   // UNICODE_TO_GBK[14826] := 16#6828;
   // UNICODE_TO_GBK[14827] := 16#96E6;
   // UNICODE_TO_GBK[14828] := 16#6829;
   // UNICODE_TO_GBK[14829] := 16#E8F2;
   // UNICODE_TO_GBK[14830] := 16#682A;
   // UNICODE_TO_GBK[14831] := 16#D6EA;
   // UNICODE_TO_GBK[14832] := 16#682B;
   // UNICODE_TO_GBK[14833] := 16#96E7;
   // UNICODE_TO_GBK[14834] := 16#682C;
   // UNICODE_TO_GBK[14835] := 16#96E8;
   // UNICODE_TO_GBK[14836] := 16#682D;
   // UNICODE_TO_GBK[14837] := 16#96E9;
   // UNICODE_TO_GBK[14838] := 16#682E;
   // UNICODE_TO_GBK[14839] := 16#96EA;
   // UNICODE_TO_GBK[14840] := 16#682F;
   // UNICODE_TO_GBK[14841] := 16#96EB;
   // UNICODE_TO_GBK[14842] := 16#6830;
   // UNICODE_TO_GBK[14843] := 16#96EC;
   // UNICODE_TO_GBK[14844] := 16#6831;
   // UNICODE_TO_GBK[14845] := 16#96ED;
   // UNICODE_TO_GBK[14846] := 16#6832;
   // UNICODE_TO_GBK[14847] := 16#E8E0;
   // UNICODE_TO_GBK[14848] := 16#6833;
   // UNICODE_TO_GBK[14849] := 16#E8E1;
   // UNICODE_TO_GBK[14850] := 16#6834;
   // UNICODE_TO_GBK[14851] := 16#96EE;
   // UNICODE_TO_GBK[14852] := 16#6835;
   // UNICODE_TO_GBK[14853] := 16#96EF;
   // UNICODE_TO_GBK[14854] := 16#6836;
   // UNICODE_TO_GBK[14855] := 16#96F0;
   // UNICODE_TO_GBK[14856] := 16#6837;
   // UNICODE_TO_GBK[14857] := 16#D1F9;
   // UNICODE_TO_GBK[14858] := 16#6838;
   // UNICODE_TO_GBK[14859] := 16#BACB;
   // UNICODE_TO_GBK[14860] := 16#6839;
   // UNICODE_TO_GBK[14861] := 16#B8F9;
   // UNICODE_TO_GBK[14862] := 16#683A;
   // UNICODE_TO_GBK[14863] := 16#96F1;
   // UNICODE_TO_GBK[14864] := 16#683B;
   // UNICODE_TO_GBK[14865] := 16#96F2;
   // UNICODE_TO_GBK[14866] := 16#683C;
   // UNICODE_TO_GBK[14867] := 16#B8F1;
   // UNICODE_TO_GBK[14868] := 16#683D;
   // UNICODE_TO_GBK[14869] := 16#D4D4;
   // UNICODE_TO_GBK[14870] := 16#683E;
   // UNICODE_TO_GBK[14871] := 16#E8EF;
   // UNICODE_TO_GBK[14872] := 16#683F;
   // UNICODE_TO_GBK[14873] := 16#96F3;
   // UNICODE_TO_GBK[14874] := 16#6840;
   // UNICODE_TO_GBK[14875] := 16#E8EE;
   // UNICODE_TO_GBK[14876] := 16#6841;
   // UNICODE_TO_GBK[14877] := 16#E8EC;
   // UNICODE_TO_GBK[14878] := 16#6842;
   // UNICODE_TO_GBK[14879] := 16#B9F0;
   // UNICODE_TO_GBK[14880] := 16#6843;
   // UNICODE_TO_GBK[14881] := 16#CCD2;
   // UNICODE_TO_GBK[14882] := 16#6844;
   // UNICODE_TO_GBK[14883] := 16#E8E6;
   // UNICODE_TO_GBK[14884] := 16#6845;
   // UNICODE_TO_GBK[14885] := 16#CEA6;
   // UNICODE_TO_GBK[14886] := 16#6846;
   // UNICODE_TO_GBK[14887] := 16#BFF2;
   // UNICODE_TO_GBK[14888] := 16#6847;
   // UNICODE_TO_GBK[14889] := 16#96F4;
   // UNICODE_TO_GBK[14890] := 16#6848;
   // UNICODE_TO_GBK[14891] := 16#B0B8;
   // UNICODE_TO_GBK[14892] := 16#6849;
   // UNICODE_TO_GBK[14893] := 16#E8F1;
   // UNICODE_TO_GBK[14894] := 16#684A;
   // UNICODE_TO_GBK[14895] := 16#E8F0;
   // UNICODE_TO_GBK[14896] := 16#684B;
   // UNICODE_TO_GBK[14897] := 16#96F5;
   // UNICODE_TO_GBK[14898] := 16#684C;
   // UNICODE_TO_GBK[14899] := 16#D7C0;
   // UNICODE_TO_GBK[14900] := 16#684D;
   // UNICODE_TO_GBK[14901] := 16#96F6;
   // UNICODE_TO_GBK[14902] := 16#684E;
   // UNICODE_TO_GBK[14903] := 16#E8E4;
   // UNICODE_TO_GBK[14904] := 16#684F;
   // UNICODE_TO_GBK[14905] := 16#96F7;
   // UNICODE_TO_GBK[14906] := 16#6850;
   // UNICODE_TO_GBK[14907] := 16#CDA9;
   // UNICODE_TO_GBK[14908] := 16#6851;
   // UNICODE_TO_GBK[14909] := 16#C9A3;
   // UNICODE_TO_GBK[14910] := 16#6852;
   // UNICODE_TO_GBK[14911] := 16#96F8;
   // UNICODE_TO_GBK[14912] := 16#6853;
   // UNICODE_TO_GBK[14913] := 16#BBB8;
   // UNICODE_TO_GBK[14914] := 16#6854;
   // UNICODE_TO_GBK[14915] := 16#BDDB;
   // UNICODE_TO_GBK[14916] := 16#6855;
   // UNICODE_TO_GBK[14917] := 16#E8EA;
   // UNICODE_TO_GBK[14918] := 16#6856;
   // UNICODE_TO_GBK[14919] := 16#96F9;
   // UNICODE_TO_GBK[14920] := 16#6857;
   // UNICODE_TO_GBK[14921] := 16#96FA;
   // UNICODE_TO_GBK[14922] := 16#6858;
   // UNICODE_TO_GBK[14923] := 16#96FB;
   // UNICODE_TO_GBK[14924] := 16#6859;
   // UNICODE_TO_GBK[14925] := 16#96FC;
   // UNICODE_TO_GBK[14926] := 16#685A;
   // UNICODE_TO_GBK[14927] := 16#96FD;
   // UNICODE_TO_GBK[14928] := 16#685B;
   // UNICODE_TO_GBK[14929] := 16#96FE;
   // UNICODE_TO_GBK[14930] := 16#685C;
   // UNICODE_TO_GBK[14931] := 16#9740;
   // UNICODE_TO_GBK[14932] := 16#685D;
   // UNICODE_TO_GBK[14933] := 16#9741;
   // UNICODE_TO_GBK[14934] := 16#685E;
   // UNICODE_TO_GBK[14935] := 16#9742;
   // UNICODE_TO_GBK[14936] := 16#685F;
   // UNICODE_TO_GBK[14937] := 16#9743;
   // UNICODE_TO_GBK[14938] := 16#6860;
   // UNICODE_TO_GBK[14939] := 16#E8E2;
   // UNICODE_TO_GBK[14940] := 16#6861;
   // UNICODE_TO_GBK[14941] := 16#E8E3;
   // UNICODE_TO_GBK[14942] := 16#6862;
   // UNICODE_TO_GBK[14943] := 16#E8E5;
   // UNICODE_TO_GBK[14944] := 16#6863;
   // UNICODE_TO_GBK[14945] := 16#B5B5;
   // UNICODE_TO_GBK[14946] := 16#6864;
   // UNICODE_TO_GBK[14947] := 16#E8E7;
   // UNICODE_TO_GBK[14948] := 16#6865;
   // UNICODE_TO_GBK[14949] := 16#C7C5;
   // UNICODE_TO_GBK[14950] := 16#6866;
   // UNICODE_TO_GBK[14951] := 16#E8EB;
   // UNICODE_TO_GBK[14952] := 16#6867;
   // UNICODE_TO_GBK[14953] := 16#E8ED;
   // UNICODE_TO_GBK[14954] := 16#6868;
   // UNICODE_TO_GBK[14955] := 16#BDB0;
   // UNICODE_TO_GBK[14956] := 16#6869;
   // UNICODE_TO_GBK[14957] := 16#D7AE;
   // UNICODE_TO_GBK[14958] := 16#686A;
   // UNICODE_TO_GBK[14959] := 16#9744;
   // UNICODE_TO_GBK[14960] := 16#686B;
   // UNICODE_TO_GBK[14961] := 16#E8F8;
   // UNICODE_TO_GBK[14962] := 16#686C;
   // UNICODE_TO_GBK[14963] := 16#9745;
   // UNICODE_TO_GBK[14964] := 16#686D;
   // UNICODE_TO_GBK[14965] := 16#9746;
   // UNICODE_TO_GBK[14966] := 16#686E;
   // UNICODE_TO_GBK[14967] := 16#9747;
   // UNICODE_TO_GBK[14968] := 16#686F;
   // UNICODE_TO_GBK[14969] := 16#9748;
   // UNICODE_TO_GBK[14970] := 16#6870;
   // UNICODE_TO_GBK[14971] := 16#9749;
   // UNICODE_TO_GBK[14972] := 16#6871;
   // UNICODE_TO_GBK[14973] := 16#974A;
   // UNICODE_TO_GBK[14974] := 16#6872;
   // UNICODE_TO_GBK[14975] := 16#974B;
   // UNICODE_TO_GBK[14976] := 16#6873;
   // UNICODE_TO_GBK[14977] := 16#974C;
   // UNICODE_TO_GBK[14978] := 16#6874;
   // UNICODE_TO_GBK[14979] := 16#E8F5;
   // UNICODE_TO_GBK[14980] := 16#6875;
   // UNICODE_TO_GBK[14981] := 16#974D;
   // UNICODE_TO_GBK[14982] := 16#6876;
   // UNICODE_TO_GBK[14983] := 16#CDB0;
   // UNICODE_TO_GBK[14984] := 16#6877;
   // UNICODE_TO_GBK[14985] := 16#E8F6;
   // UNICODE_TO_GBK[14986] := 16#6878;
   // UNICODE_TO_GBK[14987] := 16#974E;
   // UNICODE_TO_GBK[14988] := 16#6879;
   // UNICODE_TO_GBK[14989] := 16#974F;
   // UNICODE_TO_GBK[14990] := 16#687A;
   // UNICODE_TO_GBK[14991] := 16#9750;
   // UNICODE_TO_GBK[14992] := 16#687B;
   // UNICODE_TO_GBK[14993] := 16#9751;
   // UNICODE_TO_GBK[14994] := 16#687C;
   // UNICODE_TO_GBK[14995] := 16#9752;
   // UNICODE_TO_GBK[14996] := 16#687D;
   // UNICODE_TO_GBK[14997] := 16#9753;
   // UNICODE_TO_GBK[14998] := 16#687E;
   // UNICODE_TO_GBK[14999] := 16#9754;
   // UNICODE_TO_GBK[15000] := 16#687F;
   // UNICODE_TO_GBK[15001] := 16#9755;
   // UNICODE_TO_GBK[15002] := 16#6880;
   // UNICODE_TO_GBK[15003] := 16#9756;
   // UNICODE_TO_GBK[15004] := 16#6881;
   // UNICODE_TO_GBK[15005] := 16#C1BA;
   // UNICODE_TO_GBK[15006] := 16#6882;
   // UNICODE_TO_GBK[15007] := 16#9757;
   // UNICODE_TO_GBK[15008] := 16#6883;
   // UNICODE_TO_GBK[15009] := 16#E8E8;
   // UNICODE_TO_GBK[15010] := 16#6884;
   // UNICODE_TO_GBK[15011] := 16#9758;
   // UNICODE_TO_GBK[15012] := 16#6885;
   // UNICODE_TO_GBK[15013] := 16#C3B7;
   // UNICODE_TO_GBK[15014] := 16#6886;
   // UNICODE_TO_GBK[15015] := 16#B0F0;
   // UNICODE_TO_GBK[15016] := 16#6887;
   // UNICODE_TO_GBK[15017] := 16#9759;
   // UNICODE_TO_GBK[15018] := 16#6888;
   // UNICODE_TO_GBK[15019] := 16#975A;
   // UNICODE_TO_GBK[15020] := 16#6889;
   // UNICODE_TO_GBK[15021] := 16#975B;
   // UNICODE_TO_GBK[15022] := 16#688A;
   // UNICODE_TO_GBK[15023] := 16#975C;
   // UNICODE_TO_GBK[15024] := 16#688B;
   // UNICODE_TO_GBK[15025] := 16#975D;
   // UNICODE_TO_GBK[15026] := 16#688C;
   // UNICODE_TO_GBK[15027] := 16#975E;
   // UNICODE_TO_GBK[15028] := 16#688D;
   // UNICODE_TO_GBK[15029] := 16#975F;
   // UNICODE_TO_GBK[15030] := 16#688E;
   // UNICODE_TO_GBK[15031] := 16#9760;
   // UNICODE_TO_GBK[15032] := 16#688F;
   // UNICODE_TO_GBK[15033] := 16#E8F4;
   // UNICODE_TO_GBK[15034] := 16#6890;
   // UNICODE_TO_GBK[15035] := 16#9761;
   // UNICODE_TO_GBK[15036] := 16#6891;
   // UNICODE_TO_GBK[15037] := 16#9762;
   // UNICODE_TO_GBK[15038] := 16#6892;
   // UNICODE_TO_GBK[15039] := 16#9763;
   // UNICODE_TO_GBK[15040] := 16#6893;
   // UNICODE_TO_GBK[15041] := 16#E8F7;
   // UNICODE_TO_GBK[15042] := 16#6894;
   // UNICODE_TO_GBK[15043] := 16#9764;
   // UNICODE_TO_GBK[15044] := 16#6895;
   // UNICODE_TO_GBK[15045] := 16#9765;
   // UNICODE_TO_GBK[15046] := 16#6896;
   // UNICODE_TO_GBK[15047] := 16#9766;
   // UNICODE_TO_GBK[15048] := 16#6897;
   // UNICODE_TO_GBK[15049] := 16#B9A3;
   // UNICODE_TO_GBK[15050] := 16#6898;
   // UNICODE_TO_GBK[15051] := 16#9767;
   // UNICODE_TO_GBK[15052] := 16#6899;
   // UNICODE_TO_GBK[15053] := 16#9768;
   // UNICODE_TO_GBK[15054] := 16#689A;
   // UNICODE_TO_GBK[15055] := 16#9769;
   // UNICODE_TO_GBK[15056] := 16#689B;
   // UNICODE_TO_GBK[15057] := 16#976A;
   // UNICODE_TO_GBK[15058] := 16#689C;
   // UNICODE_TO_GBK[15059] := 16#976B;
   // UNICODE_TO_GBK[15060] := 16#689D;
   // UNICODE_TO_GBK[15061] := 16#976C;
   // UNICODE_TO_GBK[15062] := 16#689E;
   // UNICODE_TO_GBK[15063] := 16#976D;
   // UNICODE_TO_GBK[15064] := 16#689F;
   // UNICODE_TO_GBK[15065] := 16#976E;
   // UNICODE_TO_GBK[15066] := 16#68A0;
   // UNICODE_TO_GBK[15067] := 16#976F;
   // UNICODE_TO_GBK[15068] := 16#68A1;
   // UNICODE_TO_GBK[15069] := 16#9770;
   // UNICODE_TO_GBK[15070] := 16#68A2;
   // UNICODE_TO_GBK[15071] := 16#C9D2;
   // UNICODE_TO_GBK[15072] := 16#68A3;
   // UNICODE_TO_GBK[15073] := 16#9771;
   // UNICODE_TO_GBK[15074] := 16#68A4;
   // UNICODE_TO_GBK[15075] := 16#9772;
   // UNICODE_TO_GBK[15076] := 16#68A5;
   // UNICODE_TO_GBK[15077] := 16#9773;
   // UNICODE_TO_GBK[15078] := 16#68A6;
   // UNICODE_TO_GBK[15079] := 16#C3CE;
   // UNICODE_TO_GBK[15080] := 16#68A7;
   // UNICODE_TO_GBK[15081] := 16#CEE0;
   // UNICODE_TO_GBK[15082] := 16#68A8;
   // UNICODE_TO_GBK[15083] := 16#C0E6;
   // UNICODE_TO_GBK[15084] := 16#68A9;
   // UNICODE_TO_GBK[15085] := 16#9774;
   // UNICODE_TO_GBK[15086] := 16#68AA;
   // UNICODE_TO_GBK[15087] := 16#9775;
   // UNICODE_TO_GBK[15088] := 16#68AB;
   // UNICODE_TO_GBK[15089] := 16#9776;
   // UNICODE_TO_GBK[15090] := 16#68AC;
   // UNICODE_TO_GBK[15091] := 16#9777;
   // UNICODE_TO_GBK[15092] := 16#68AD;
   // UNICODE_TO_GBK[15093] := 16#CBF3;
   // UNICODE_TO_GBK[15094] := 16#68AE;
   // UNICODE_TO_GBK[15095] := 16#9778;
   // UNICODE_TO_GBK[15096] := 16#68AF;
   // UNICODE_TO_GBK[15097] := 16#CCDD;
   // UNICODE_TO_GBK[15098] := 16#68B0;
   // UNICODE_TO_GBK[15099] := 16#D0B5;
   // UNICODE_TO_GBK[15100] := 16#68B1;
   // UNICODE_TO_GBK[15101] := 16#9779;
   // UNICODE_TO_GBK[15102] := 16#68B2;
   // UNICODE_TO_GBK[15103] := 16#977A;
   // UNICODE_TO_GBK[15104] := 16#68B3;
   // UNICODE_TO_GBK[15105] := 16#CAE1;
   // UNICODE_TO_GBK[15106] := 16#68B4;
   // UNICODE_TO_GBK[15107] := 16#977B;
   // UNICODE_TO_GBK[15108] := 16#68B5;
   // UNICODE_TO_GBK[15109] := 16#E8F3;
   // UNICODE_TO_GBK[15110] := 16#68B6;
   // UNICODE_TO_GBK[15111] := 16#977C;
   // UNICODE_TO_GBK[15112] := 16#68B7;
   // UNICODE_TO_GBK[15113] := 16#977D;
   // UNICODE_TO_GBK[15114] := 16#68B8;
   // UNICODE_TO_GBK[15115] := 16#977E;
   // UNICODE_TO_GBK[15116] := 16#68B9;
   // UNICODE_TO_GBK[15117] := 16#9780;
   // UNICODE_TO_GBK[15118] := 16#68BA;
   // UNICODE_TO_GBK[15119] := 16#9781;
   // UNICODE_TO_GBK[15120] := 16#68BB;
   // UNICODE_TO_GBK[15121] := 16#9782;
   // UNICODE_TO_GBK[15122] := 16#68BC;
   // UNICODE_TO_GBK[15123] := 16#9783;
   // UNICODE_TO_GBK[15124] := 16#68BD;
   // UNICODE_TO_GBK[15125] := 16#9784;
   // UNICODE_TO_GBK[15126] := 16#68BE;
   // UNICODE_TO_GBK[15127] := 16#9785;
   // UNICODE_TO_GBK[15128] := 16#68BF;
   // UNICODE_TO_GBK[15129] := 16#9786;
   // UNICODE_TO_GBK[15130] := 16#68C0;
   // UNICODE_TO_GBK[15131] := 16#BCEC;
   // UNICODE_TO_GBK[15132] := 16#68C1;
   // UNICODE_TO_GBK[15133] := 16#9787;
   // UNICODE_TO_GBK[15134] := 16#68C2;
   // UNICODE_TO_GBK[15135] := 16#E8F9;
   // UNICODE_TO_GBK[15136] := 16#68C3;
   // UNICODE_TO_GBK[15137] := 16#9788;
   // UNICODE_TO_GBK[15138] := 16#68C4;
   // UNICODE_TO_GBK[15139] := 16#9789;
   // UNICODE_TO_GBK[15140] := 16#68C5;
   // UNICODE_TO_GBK[15141] := 16#978A;
   // UNICODE_TO_GBK[15142] := 16#68C6;
   // UNICODE_TO_GBK[15143] := 16#978B;
   // UNICODE_TO_GBK[15144] := 16#68C7;
   // UNICODE_TO_GBK[15145] := 16#978C;
   // UNICODE_TO_GBK[15146] := 16#68C8;
   // UNICODE_TO_GBK[15147] := 16#978D;
   // UNICODE_TO_GBK[15148] := 16#68C9;
   // UNICODE_TO_GBK[15149] := 16#C3DE;
   // UNICODE_TO_GBK[15150] := 16#68CA;
   // UNICODE_TO_GBK[15151] := 16#978E;
   // UNICODE_TO_GBK[15152] := 16#68CB;
   // UNICODE_TO_GBK[15153] := 16#C6E5;
   // UNICODE_TO_GBK[15154] := 16#68CC;
   // UNICODE_TO_GBK[15155] := 16#978F;
   // UNICODE_TO_GBK[15156] := 16#68CD;
   // UNICODE_TO_GBK[15157] := 16#B9F7;
   // UNICODE_TO_GBK[15158] := 16#68CE;
   // UNICODE_TO_GBK[15159] := 16#9790;
   // UNICODE_TO_GBK[15160] := 16#68CF;
   // UNICODE_TO_GBK[15161] := 16#9791;
   // UNICODE_TO_GBK[15162] := 16#68D0;
   // UNICODE_TO_GBK[15163] := 16#9792;
   // UNICODE_TO_GBK[15164] := 16#68D1;
   // UNICODE_TO_GBK[15165] := 16#9793;
   // UNICODE_TO_GBK[15166] := 16#68D2;
   // UNICODE_TO_GBK[15167] := 16#B0F4;
   // UNICODE_TO_GBK[15168] := 16#68D3;
   // UNICODE_TO_GBK[15169] := 16#9794;
   // UNICODE_TO_GBK[15170] := 16#68D4;
   // UNICODE_TO_GBK[15171] := 16#9795;
   // UNICODE_TO_GBK[15172] := 16#68D5;
   // UNICODE_TO_GBK[15173] := 16#D7D8;
   // UNICODE_TO_GBK[15174] := 16#68D6;
   // UNICODE_TO_GBK[15175] := 16#9796;
   // UNICODE_TO_GBK[15176] := 16#68D7;
   // UNICODE_TO_GBK[15177] := 16#9797;
   // UNICODE_TO_GBK[15178] := 16#68D8;
   // UNICODE_TO_GBK[15179] := 16#BCAC;
   // UNICODE_TO_GBK[15180] := 16#68D9;
   // UNICODE_TO_GBK[15181] := 16#9798;
   // UNICODE_TO_GBK[15182] := 16#68DA;
   // UNICODE_TO_GBK[15183] := 16#C5EF;
   // UNICODE_TO_GBK[15184] := 16#68DB;
   // UNICODE_TO_GBK[15185] := 16#9799;
   // UNICODE_TO_GBK[15186] := 16#68DC;
   // UNICODE_TO_GBK[15187] := 16#979A;
   // UNICODE_TO_GBK[15188] := 16#68DD;
   // UNICODE_TO_GBK[15189] := 16#979B;
   // UNICODE_TO_GBK[15190] := 16#68DE;
   // UNICODE_TO_GBK[15191] := 16#979C;
   // UNICODE_TO_GBK[15192] := 16#68DF;
   // UNICODE_TO_GBK[15193] := 16#979D;
   // UNICODE_TO_GBK[15194] := 16#68E0;
   // UNICODE_TO_GBK[15195] := 16#CCC4;
   // UNICODE_TO_GBK[15196] := 16#68E1;
   // UNICODE_TO_GBK[15197] := 16#979E;
   // UNICODE_TO_GBK[15198] := 16#68E2;
   // UNICODE_TO_GBK[15199] := 16#979F;
   // UNICODE_TO_GBK[15200] := 16#68E3;
   // UNICODE_TO_GBK[15201] := 16#E9A6;
   // UNICODE_TO_GBK[15202] := 16#68E4;
   // UNICODE_TO_GBK[15203] := 16#97A0;
   // UNICODE_TO_GBK[15204] := 16#68E5;
   // UNICODE_TO_GBK[15205] := 16#97A1;
   // UNICODE_TO_GBK[15206] := 16#68E6;
   // UNICODE_TO_GBK[15207] := 16#97A2;
   // UNICODE_TO_GBK[15208] := 16#68E7;
   // UNICODE_TO_GBK[15209] := 16#97A3;
   // UNICODE_TO_GBK[15210] := 16#68E8;
   // UNICODE_TO_GBK[15211] := 16#97A4;
   // UNICODE_TO_GBK[15212] := 16#68E9;
   // UNICODE_TO_GBK[15213] := 16#97A5;
   // UNICODE_TO_GBK[15214] := 16#68EA;
   // UNICODE_TO_GBK[15215] := 16#97A6;
   // UNICODE_TO_GBK[15216] := 16#68EB;
   // UNICODE_TO_GBK[15217] := 16#97A7;
   // UNICODE_TO_GBK[15218] := 16#68EC;
   // UNICODE_TO_GBK[15219] := 16#97A8;
   // UNICODE_TO_GBK[15220] := 16#68ED;
   // UNICODE_TO_GBK[15221] := 16#97A9;
   // UNICODE_TO_GBK[15222] := 16#68EE;
   // UNICODE_TO_GBK[15223] := 16#C9AD;
   // UNICODE_TO_GBK[15224] := 16#68EF;
   // UNICODE_TO_GBK[15225] := 16#97AA;
   // UNICODE_TO_GBK[15226] := 16#68F0;
   // UNICODE_TO_GBK[15227] := 16#E9A2;
   // UNICODE_TO_GBK[15228] := 16#68F1;
   // UNICODE_TO_GBK[15229] := 16#C0E2;
   // UNICODE_TO_GBK[15230] := 16#68F2;
   // UNICODE_TO_GBK[15231] := 16#97AB;
   // UNICODE_TO_GBK[15232] := 16#68F3;
   // UNICODE_TO_GBK[15233] := 16#97AC;
   // UNICODE_TO_GBK[15234] := 16#68F4;
   // UNICODE_TO_GBK[15235] := 16#97AD;
   // UNICODE_TO_GBK[15236] := 16#68F5;
   // UNICODE_TO_GBK[15237] := 16#BFC3;
   // UNICODE_TO_GBK[15238] := 16#68F6;
   // UNICODE_TO_GBK[15239] := 16#97AE;
   // UNICODE_TO_GBK[15240] := 16#68F7;
   // UNICODE_TO_GBK[15241] := 16#97AF;
   // UNICODE_TO_GBK[15242] := 16#68F8;
   // UNICODE_TO_GBK[15243] := 16#97B0;
   // UNICODE_TO_GBK[15244] := 16#68F9;
   // UNICODE_TO_GBK[15245] := 16#E8FE;
   // UNICODE_TO_GBK[15246] := 16#68FA;
   // UNICODE_TO_GBK[15247] := 16#B9D7;
   // UNICODE_TO_GBK[15248] := 16#68FB;
   // UNICODE_TO_GBK[15249] := 16#97B1;
   // UNICODE_TO_GBK[15250] := 16#68FC;
   // UNICODE_TO_GBK[15251] := 16#E8FB;
   // UNICODE_TO_GBK[15252] := 16#68FD;
   // UNICODE_TO_GBK[15253] := 16#97B2;
   // UNICODE_TO_GBK[15254] := 16#68FE;
   // UNICODE_TO_GBK[15255] := 16#97B3;
   // UNICODE_TO_GBK[15256] := 16#68FF;
   // UNICODE_TO_GBK[15257] := 16#97B4;
   // UNICODE_TO_GBK[15258] := 16#6900;
   // UNICODE_TO_GBK[15259] := 16#97B5;
   // UNICODE_TO_GBK[15260] := 16#6901;
   // UNICODE_TO_GBK[15261] := 16#E9A4;
   // UNICODE_TO_GBK[15262] := 16#6902;
   // UNICODE_TO_GBK[15263] := 16#97B6;
   // UNICODE_TO_GBK[15264] := 16#6903;
   // UNICODE_TO_GBK[15265] := 16#97B7;
   // UNICODE_TO_GBK[15266] := 16#6904;
   // UNICODE_TO_GBK[15267] := 16#97B8;
   // UNICODE_TO_GBK[15268] := 16#6905;
   // UNICODE_TO_GBK[15269] := 16#D2CE;
   // UNICODE_TO_GBK[15270] := 16#6906;
   // UNICODE_TO_GBK[15271] := 16#97B9;
   // UNICODE_TO_GBK[15272] := 16#6907;
   // UNICODE_TO_GBK[15273] := 16#97BA;
   // UNICODE_TO_GBK[15274] := 16#6908;
   // UNICODE_TO_GBK[15275] := 16#97BB;
   // UNICODE_TO_GBK[15276] := 16#6909;
   // UNICODE_TO_GBK[15277] := 16#97BC;
   // UNICODE_TO_GBK[15278] := 16#690A;
   // UNICODE_TO_GBK[15279] := 16#97BD;
   // UNICODE_TO_GBK[15280] := 16#690B;
   // UNICODE_TO_GBK[15281] := 16#E9A3;
   // UNICODE_TO_GBK[15282] := 16#690C;
   // UNICODE_TO_GBK[15283] := 16#97BE;
   // UNICODE_TO_GBK[15284] := 16#690D;
   // UNICODE_TO_GBK[15285] := 16#D6B2;
   // UNICODE_TO_GBK[15286] := 16#690E;
   // UNICODE_TO_GBK[15287] := 16#D7B5;
   // UNICODE_TO_GBK[15288] := 16#690F;
   // UNICODE_TO_GBK[15289] := 16#97BF;
   // UNICODE_TO_GBK[15290] := 16#6910;
   // UNICODE_TO_GBK[15291] := 16#E9A7;
   // UNICODE_TO_GBK[15292] := 16#6911;
   // UNICODE_TO_GBK[15293] := 16#97C0;
   // UNICODE_TO_GBK[15294] := 16#6912;
   // UNICODE_TO_GBK[15295] := 16#BDB7;
   // UNICODE_TO_GBK[15296] := 16#6913;
   // UNICODE_TO_GBK[15297] := 16#97C1;
   // UNICODE_TO_GBK[15298] := 16#6914;
   // UNICODE_TO_GBK[15299] := 16#97C2;
   // UNICODE_TO_GBK[15300] := 16#6915;
   // UNICODE_TO_GBK[15301] := 16#97C3;
   // UNICODE_TO_GBK[15302] := 16#6916;
   // UNICODE_TO_GBK[15303] := 16#97C4;
   // UNICODE_TO_GBK[15304] := 16#6917;
   // UNICODE_TO_GBK[15305] := 16#97C5;
   // UNICODE_TO_GBK[15306] := 16#6918;
   // UNICODE_TO_GBK[15307] := 16#97C6;
   // UNICODE_TO_GBK[15308] := 16#6919;
   // UNICODE_TO_GBK[15309] := 16#97C7;
   // UNICODE_TO_GBK[15310] := 16#691A;
   // UNICODE_TO_GBK[15311] := 16#97C8;
   // UNICODE_TO_GBK[15312] := 16#691B;
   // UNICODE_TO_GBK[15313] := 16#97C9;
   // UNICODE_TO_GBK[15314] := 16#691C;
   // UNICODE_TO_GBK[15315] := 16#97CA;
   // UNICODE_TO_GBK[15316] := 16#691D;
   // UNICODE_TO_GBK[15317] := 16#97CB;
   // UNICODE_TO_GBK[15318] := 16#691E;
   // UNICODE_TO_GBK[15319] := 16#97CC;
   // UNICODE_TO_GBK[15320] := 16#691F;
   // UNICODE_TO_GBK[15321] := 16#E8FC;
   // UNICODE_TO_GBK[15322] := 16#6920;
   // UNICODE_TO_GBK[15323] := 16#E8FD;
   // UNICODE_TO_GBK[15324] := 16#6921;
   // UNICODE_TO_GBK[15325] := 16#97CD;
   // UNICODE_TO_GBK[15326] := 16#6922;
   // UNICODE_TO_GBK[15327] := 16#97CE;
   // UNICODE_TO_GBK[15328] := 16#6923;
   // UNICODE_TO_GBK[15329] := 16#97CF;
   // UNICODE_TO_GBK[15330] := 16#6924;
   // UNICODE_TO_GBK[15331] := 16#E9A1;
   // UNICODE_TO_GBK[15332] := 16#6925;
   // UNICODE_TO_GBK[15333] := 16#97D0;
   // UNICODE_TO_GBK[15334] := 16#6926;
   // UNICODE_TO_GBK[15335] := 16#97D1;
   // UNICODE_TO_GBK[15336] := 16#6927;
   // UNICODE_TO_GBK[15337] := 16#97D2;
   // UNICODE_TO_GBK[15338] := 16#6928;
   // UNICODE_TO_GBK[15339] := 16#97D3;
   // UNICODE_TO_GBK[15340] := 16#6929;
   // UNICODE_TO_GBK[15341] := 16#97D4;
   // UNICODE_TO_GBK[15342] := 16#692A;
   // UNICODE_TO_GBK[15343] := 16#97D5;
   // UNICODE_TO_GBK[15344] := 16#692B;
   // UNICODE_TO_GBK[15345] := 16#97D6;
   // UNICODE_TO_GBK[15346] := 16#692C;
   // UNICODE_TO_GBK[15347] := 16#97D7;
   // UNICODE_TO_GBK[15348] := 16#692D;
   // UNICODE_TO_GBK[15349] := 16#CDD6;
   // UNICODE_TO_GBK[15350] := 16#692E;
   // UNICODE_TO_GBK[15351] := 16#97D8;
   // UNICODE_TO_GBK[15352] := 16#692F;
   // UNICODE_TO_GBK[15353] := 16#97D9;
   // UNICODE_TO_GBK[15354] := 16#6930;
   // UNICODE_TO_GBK[15355] := 16#D2AC;
   // UNICODE_TO_GBK[15356] := 16#6931;
   // UNICODE_TO_GBK[15357] := 16#97DA;
   // UNICODE_TO_GBK[15358] := 16#6932;
   // UNICODE_TO_GBK[15359] := 16#97DB;
   // UNICODE_TO_GBK[15360] := 16#6933;
   // UNICODE_TO_GBK[15361] := 16#97DC;
   // UNICODE_TO_GBK[15362] := 16#6934;
   // UNICODE_TO_GBK[15363] := 16#E9B2;
   // UNICODE_TO_GBK[15364] := 16#6935;
   // UNICODE_TO_GBK[15365] := 16#97DD;
   // UNICODE_TO_GBK[15366] := 16#6936;
   // UNICODE_TO_GBK[15367] := 16#97DE;
   // UNICODE_TO_GBK[15368] := 16#6937;
   // UNICODE_TO_GBK[15369] := 16#97DF;
   // UNICODE_TO_GBK[15370] := 16#6938;
   // UNICODE_TO_GBK[15371] := 16#97E0;
   // UNICODE_TO_GBK[15372] := 16#6939;
   // UNICODE_TO_GBK[15373] := 16#E9A9;
   // UNICODE_TO_GBK[15374] := 16#693A;
   // UNICODE_TO_GBK[15375] := 16#97E1;
   // UNICODE_TO_GBK[15376] := 16#693B;
   // UNICODE_TO_GBK[15377] := 16#97E2;
   // UNICODE_TO_GBK[15378] := 16#693C;
   // UNICODE_TO_GBK[15379] := 16#97E3;
   // UNICODE_TO_GBK[15380] := 16#693D;
   // UNICODE_TO_GBK[15381] := 16#B4AA;
   // UNICODE_TO_GBK[15382] := 16#693E;
   // UNICODE_TO_GBK[15383] := 16#97E4;
   // UNICODE_TO_GBK[15384] := 16#693F;
   // UNICODE_TO_GBK[15385] := 16#B4BB;
   // UNICODE_TO_GBK[15386] := 16#6940;
   // UNICODE_TO_GBK[15387] := 16#97E5;
   // UNICODE_TO_GBK[15388] := 16#6941;
   // UNICODE_TO_GBK[15389] := 16#97E6;
   // UNICODE_TO_GBK[15390] := 16#6942;
   // UNICODE_TO_GBK[15391] := 16#E9AB;
   // UNICODE_TO_GBK[15392] := 16#6943;
   // UNICODE_TO_GBK[15393] := 16#97E7;
   // UNICODE_TO_GBK[15394] := 16#6944;
   // UNICODE_TO_GBK[15395] := 16#97E8;
   // UNICODE_TO_GBK[15396] := 16#6945;
   // UNICODE_TO_GBK[15397] := 16#97E9;
   // UNICODE_TO_GBK[15398] := 16#6946;
   // UNICODE_TO_GBK[15399] := 16#97EA;
   // UNICODE_TO_GBK[15400] := 16#6947;
   // UNICODE_TO_GBK[15401] := 16#97EB;
   // UNICODE_TO_GBK[15402] := 16#6948;
   // UNICODE_TO_GBK[15403] := 16#97EC;
   // UNICODE_TO_GBK[15404] := 16#6949;
   // UNICODE_TO_GBK[15405] := 16#97ED;
   // UNICODE_TO_GBK[15406] := 16#694A;
   // UNICODE_TO_GBK[15407] := 16#97EE;
   // UNICODE_TO_GBK[15408] := 16#694B;
   // UNICODE_TO_GBK[15409] := 16#97EF;
   // UNICODE_TO_GBK[15410] := 16#694C;
   // UNICODE_TO_GBK[15411] := 16#97F0;
   // UNICODE_TO_GBK[15412] := 16#694D;
   // UNICODE_TO_GBK[15413] := 16#97F1;
   // UNICODE_TO_GBK[15414] := 16#694E;
   // UNICODE_TO_GBK[15415] := 16#97F2;
   // UNICODE_TO_GBK[15416] := 16#694F;
   // UNICODE_TO_GBK[15417] := 16#97F3;
   // UNICODE_TO_GBK[15418] := 16#6950;
   // UNICODE_TO_GBK[15419] := 16#97F4;
   // UNICODE_TO_GBK[15420] := 16#6951;
   // UNICODE_TO_GBK[15421] := 16#97F5;
   // UNICODE_TO_GBK[15422] := 16#6952;
   // UNICODE_TO_GBK[15423] := 16#97F6;
   // UNICODE_TO_GBK[15424] := 16#6953;
   // UNICODE_TO_GBK[15425] := 16#97F7;
   // UNICODE_TO_GBK[15426] := 16#6954;
   // UNICODE_TO_GBK[15427] := 16#D0A8;
   // UNICODE_TO_GBK[15428] := 16#6955;
   // UNICODE_TO_GBK[15429] := 16#97F8;
   // UNICODE_TO_GBK[15430] := 16#6956;
   // UNICODE_TO_GBK[15431] := 16#97F9;
   // UNICODE_TO_GBK[15432] := 16#6957;
   // UNICODE_TO_GBK[15433] := 16#E9A5;
   // UNICODE_TO_GBK[15434] := 16#6958;
   // UNICODE_TO_GBK[15435] := 16#97FA;
   // UNICODE_TO_GBK[15436] := 16#6959;
   // UNICODE_TO_GBK[15437] := 16#97FB;
   // UNICODE_TO_GBK[15438] := 16#695A;
   // UNICODE_TO_GBK[15439] := 16#B3FE;
   // UNICODE_TO_GBK[15440] := 16#695B;
   // UNICODE_TO_GBK[15441] := 16#97FC;
   // UNICODE_TO_GBK[15442] := 16#695C;
   // UNICODE_TO_GBK[15443] := 16#97FD;
   // UNICODE_TO_GBK[15444] := 16#695D;
   // UNICODE_TO_GBK[15445] := 16#E9AC;
   // UNICODE_TO_GBK[15446] := 16#695E;
   // UNICODE_TO_GBK[15447] := 16#C0E3;
   // UNICODE_TO_GBK[15448] := 16#695F;
   // UNICODE_TO_GBK[15449] := 16#97FE;
   // UNICODE_TO_GBK[15450] := 16#6960;
   // UNICODE_TO_GBK[15451] := 16#E9AA;
   // UNICODE_TO_GBK[15452] := 16#6961;
   // UNICODE_TO_GBK[15453] := 16#9840;
   // UNICODE_TO_GBK[15454] := 16#6962;
   // UNICODE_TO_GBK[15455] := 16#9841;
   // UNICODE_TO_GBK[15456] := 16#6963;
   // UNICODE_TO_GBK[15457] := 16#E9B9;
   // UNICODE_TO_GBK[15458] := 16#6964;
   // UNICODE_TO_GBK[15459] := 16#9842;
   // UNICODE_TO_GBK[15460] := 16#6965;
   // UNICODE_TO_GBK[15461] := 16#9843;
   // UNICODE_TO_GBK[15462] := 16#6966;
   // UNICODE_TO_GBK[15463] := 16#E9B8;
   // UNICODE_TO_GBK[15464] := 16#6967;
   // UNICODE_TO_GBK[15465] := 16#9844;
   // UNICODE_TO_GBK[15466] := 16#6968;
   // UNICODE_TO_GBK[15467] := 16#9845;
   // UNICODE_TO_GBK[15468] := 16#6969;
   // UNICODE_TO_GBK[15469] := 16#9846;
   // UNICODE_TO_GBK[15470] := 16#696A;
   // UNICODE_TO_GBK[15471] := 16#9847;
   // UNICODE_TO_GBK[15472] := 16#696B;
   // UNICODE_TO_GBK[15473] := 16#E9AE;
   // UNICODE_TO_GBK[15474] := 16#696C;
   // UNICODE_TO_GBK[15475] := 16#9848;
   // UNICODE_TO_GBK[15476] := 16#696D;
   // UNICODE_TO_GBK[15477] := 16#9849;
   // UNICODE_TO_GBK[15478] := 16#696E;
   // UNICODE_TO_GBK[15479] := 16#E8FA;
   // UNICODE_TO_GBK[15480] := 16#696F;
   // UNICODE_TO_GBK[15481] := 16#984A;
   // UNICODE_TO_GBK[15482] := 16#6970;
   // UNICODE_TO_GBK[15483] := 16#984B;
   // UNICODE_TO_GBK[15484] := 16#6971;
   // UNICODE_TO_GBK[15485] := 16#E9A8;
   // UNICODE_TO_GBK[15486] := 16#6972;
   // UNICODE_TO_GBK[15487] := 16#984C;
   // UNICODE_TO_GBK[15488] := 16#6973;
   // UNICODE_TO_GBK[15489] := 16#984D;
   // UNICODE_TO_GBK[15490] := 16#6974;
   // UNICODE_TO_GBK[15491] := 16#984E;
   // UNICODE_TO_GBK[15492] := 16#6975;
   // UNICODE_TO_GBK[15493] := 16#984F;
   // UNICODE_TO_GBK[15494] := 16#6976;
   // UNICODE_TO_GBK[15495] := 16#9850;
   // UNICODE_TO_GBK[15496] := 16#6977;
   // UNICODE_TO_GBK[15497] := 16#BFAC;
   // UNICODE_TO_GBK[15498] := 16#6978;
   // UNICODE_TO_GBK[15499] := 16#E9B1;
   // UNICODE_TO_GBK[15500] := 16#6979;
   // UNICODE_TO_GBK[15501] := 16#E9BA;
   // UNICODE_TO_GBK[15502] := 16#697A;
   // UNICODE_TO_GBK[15503] := 16#9851;
   // UNICODE_TO_GBK[15504] := 16#697B;
   // UNICODE_TO_GBK[15505] := 16#9852;
   // UNICODE_TO_GBK[15506] := 16#697C;
   // UNICODE_TO_GBK[15507] := 16#C2A5;
   // UNICODE_TO_GBK[15508] := 16#697D;
   // UNICODE_TO_GBK[15509] := 16#9853;
   // UNICODE_TO_GBK[15510] := 16#697E;
   // UNICODE_TO_GBK[15511] := 16#9854;
   // UNICODE_TO_GBK[15512] := 16#697F;
   // UNICODE_TO_GBK[15513] := 16#9855;
   // UNICODE_TO_GBK[15514] := 16#6980;
   // UNICODE_TO_GBK[15515] := 16#E9AF;
   // UNICODE_TO_GBK[15516] := 16#6981;
   // UNICODE_TO_GBK[15517] := 16#9856;
   // UNICODE_TO_GBK[15518] := 16#6982;
   // UNICODE_TO_GBK[15519] := 16#B8C5;
   // UNICODE_TO_GBK[15520] := 16#6983;
   // UNICODE_TO_GBK[15521] := 16#9857;
   // UNICODE_TO_GBK[15522] := 16#6984;
   // UNICODE_TO_GBK[15523] := 16#E9AD;
   // UNICODE_TO_GBK[15524] := 16#6985;
   // UNICODE_TO_GBK[15525] := 16#9858;
   // UNICODE_TO_GBK[15526] := 16#6986;
   // UNICODE_TO_GBK[15527] := 16#D3DC;
   // UNICODE_TO_GBK[15528] := 16#6987;
   // UNICODE_TO_GBK[15529] := 16#E9B4;
   // UNICODE_TO_GBK[15530] := 16#6988;
   // UNICODE_TO_GBK[15531] := 16#E9B5;
   // UNICODE_TO_GBK[15532] := 16#6989;
   // UNICODE_TO_GBK[15533] := 16#E9B7;
   // UNICODE_TO_GBK[15534] := 16#698A;
   // UNICODE_TO_GBK[15535] := 16#9859;
   // UNICODE_TO_GBK[15536] := 16#698B;
   // UNICODE_TO_GBK[15537] := 16#985A;
   // UNICODE_TO_GBK[15538] := 16#698C;
   // UNICODE_TO_GBK[15539] := 16#985B;
   // UNICODE_TO_GBK[15540] := 16#698D;
   // UNICODE_TO_GBK[15541] := 16#E9C7;
   // UNICODE_TO_GBK[15542] := 16#698E;
   // UNICODE_TO_GBK[15543] := 16#985C;
   // UNICODE_TO_GBK[15544] := 16#698F;
   // UNICODE_TO_GBK[15545] := 16#985D;
   // UNICODE_TO_GBK[15546] := 16#6990;
   // UNICODE_TO_GBK[15547] := 16#985E;
   // UNICODE_TO_GBK[15548] := 16#6991;
   // UNICODE_TO_GBK[15549] := 16#985F;
   // UNICODE_TO_GBK[15550] := 16#6992;
   // UNICODE_TO_GBK[15551] := 16#9860;
   // UNICODE_TO_GBK[15552] := 16#6993;
   // UNICODE_TO_GBK[15553] := 16#9861;
   // UNICODE_TO_GBK[15554] := 16#6994;
   // UNICODE_TO_GBK[15555] := 16#C0C6;
   // UNICODE_TO_GBK[15556] := 16#6995;
   // UNICODE_TO_GBK[15557] := 16#E9C5;
   // UNICODE_TO_GBK[15558] := 16#6996;
   // UNICODE_TO_GBK[15559] := 16#9862;
   // UNICODE_TO_GBK[15560] := 16#6997;
   // UNICODE_TO_GBK[15561] := 16#9863;
   // UNICODE_TO_GBK[15562] := 16#6998;
   // UNICODE_TO_GBK[15563] := 16#E9B0;
   // UNICODE_TO_GBK[15564] := 16#6999;
   // UNICODE_TO_GBK[15565] := 16#9864;
   // UNICODE_TO_GBK[15566] := 16#699A;
   // UNICODE_TO_GBK[15567] := 16#9865;
   // UNICODE_TO_GBK[15568] := 16#699B;
   // UNICODE_TO_GBK[15569] := 16#E9BB;
   // UNICODE_TO_GBK[15570] := 16#699C;
   // UNICODE_TO_GBK[15571] := 16#B0F1;
   // UNICODE_TO_GBK[15572] := 16#699D;
   // UNICODE_TO_GBK[15573] := 16#9866;
   // UNICODE_TO_GBK[15574] := 16#699E;
   // UNICODE_TO_GBK[15575] := 16#9867;
   // UNICODE_TO_GBK[15576] := 16#699F;
   // UNICODE_TO_GBK[15577] := 16#9868;
   // UNICODE_TO_GBK[15578] := 16#69A0;
   // UNICODE_TO_GBK[15579] := 16#9869;
   // UNICODE_TO_GBK[15580] := 16#69A1;
   // UNICODE_TO_GBK[15581] := 16#986A;
   // UNICODE_TO_GBK[15582] := 16#69A2;
   // UNICODE_TO_GBK[15583] := 16#986B;
   // UNICODE_TO_GBK[15584] := 16#69A3;
   // UNICODE_TO_GBK[15585] := 16#986C;
   // UNICODE_TO_GBK[15586] := 16#69A4;
   // UNICODE_TO_GBK[15587] := 16#986D;
   // UNICODE_TO_GBK[15588] := 16#69A5;
   // UNICODE_TO_GBK[15589] := 16#986E;
   // UNICODE_TO_GBK[15590] := 16#69A6;
   // UNICODE_TO_GBK[15591] := 16#986F;
   // UNICODE_TO_GBK[15592] := 16#69A7;
   // UNICODE_TO_GBK[15593] := 16#E9BC;
   // UNICODE_TO_GBK[15594] := 16#69A8;
   // UNICODE_TO_GBK[15595] := 16#D5A5;
   // UNICODE_TO_GBK[15596] := 16#69A9;
   // UNICODE_TO_GBK[15597] := 16#9870;
   // UNICODE_TO_GBK[15598] := 16#69AA;
   // UNICODE_TO_GBK[15599] := 16#9871;
   // UNICODE_TO_GBK[15600] := 16#69AB;
   // UNICODE_TO_GBK[15601] := 16#E9BE;
   // UNICODE_TO_GBK[15602] := 16#69AC;
   // UNICODE_TO_GBK[15603] := 16#9872;
   // UNICODE_TO_GBK[15604] := 16#69AD;
   // UNICODE_TO_GBK[15605] := 16#E9BF;
   // UNICODE_TO_GBK[15606] := 16#69AE;
   // UNICODE_TO_GBK[15607] := 16#9873;
   // UNICODE_TO_GBK[15608] := 16#69AF;
   // UNICODE_TO_GBK[15609] := 16#9874;
   // UNICODE_TO_GBK[15610] := 16#69B0;
   // UNICODE_TO_GBK[15611] := 16#9875;
   // UNICODE_TO_GBK[15612] := 16#69B1;
   // UNICODE_TO_GBK[15613] := 16#E9C1;
   // UNICODE_TO_GBK[15614] := 16#69B2;
   // UNICODE_TO_GBK[15615] := 16#9876;
   // UNICODE_TO_GBK[15616] := 16#69B3;
   // UNICODE_TO_GBK[15617] := 16#9877;
   // UNICODE_TO_GBK[15618] := 16#69B4;
   // UNICODE_TO_GBK[15619] := 16#C1F1;
   // UNICODE_TO_GBK[15620] := 16#69B5;
   // UNICODE_TO_GBK[15621] := 16#9878;
   // UNICODE_TO_GBK[15622] := 16#69B6;
   // UNICODE_TO_GBK[15623] := 16#9879;
   // UNICODE_TO_GBK[15624] := 16#69B7;
   // UNICODE_TO_GBK[15625] := 16#C8B6;
   // UNICODE_TO_GBK[15626] := 16#69B8;
   // UNICODE_TO_GBK[15627] := 16#987A;
   // UNICODE_TO_GBK[15628] := 16#69B9;
   // UNICODE_TO_GBK[15629] := 16#987B;
   // UNICODE_TO_GBK[15630] := 16#69BA;
   // UNICODE_TO_GBK[15631] := 16#987C;
   // UNICODE_TO_GBK[15632] := 16#69BB;
   // UNICODE_TO_GBK[15633] := 16#E9BD;
   // UNICODE_TO_GBK[15634] := 16#69BC;
   // UNICODE_TO_GBK[15635] := 16#987D;
   // UNICODE_TO_GBK[15636] := 16#69BD;
   // UNICODE_TO_GBK[15637] := 16#987E;
   // UNICODE_TO_GBK[15638] := 16#69BE;
   // UNICODE_TO_GBK[15639] := 16#9880;
   // UNICODE_TO_GBK[15640] := 16#69BF;
   // UNICODE_TO_GBK[15641] := 16#9881;
   // UNICODE_TO_GBK[15642] := 16#69C0;
   // UNICODE_TO_GBK[15643] := 16#9882;
   // UNICODE_TO_GBK[15644] := 16#69C1;
   // UNICODE_TO_GBK[15645] := 16#E9C2;
   // UNICODE_TO_GBK[15646] := 16#69C2;
   // UNICODE_TO_GBK[15647] := 16#9883;
   // UNICODE_TO_GBK[15648] := 16#69C3;
   // UNICODE_TO_GBK[15649] := 16#9884;
   // UNICODE_TO_GBK[15650] := 16#69C4;
   // UNICODE_TO_GBK[15651] := 16#9885;
   // UNICODE_TO_GBK[15652] := 16#69C5;
   // UNICODE_TO_GBK[15653] := 16#9886;
   // UNICODE_TO_GBK[15654] := 16#69C6;
   // UNICODE_TO_GBK[15655] := 16#9887;
   // UNICODE_TO_GBK[15656] := 16#69C7;
   // UNICODE_TO_GBK[15657] := 16#9888;
   // UNICODE_TO_GBK[15658] := 16#69C8;
   // UNICODE_TO_GBK[15659] := 16#9889;
   // UNICODE_TO_GBK[15660] := 16#69C9;
   // UNICODE_TO_GBK[15661] := 16#988A;
   // UNICODE_TO_GBK[15662] := 16#69CA;
   // UNICODE_TO_GBK[15663] := 16#E9C3;
   // UNICODE_TO_GBK[15664] := 16#69CB;
   // UNICODE_TO_GBK[15665] := 16#988B;
   // UNICODE_TO_GBK[15666] := 16#69CC;
   // UNICODE_TO_GBK[15667] := 16#E9B3;
   // UNICODE_TO_GBK[15668] := 16#69CD;
   // UNICODE_TO_GBK[15669] := 16#988C;
   // UNICODE_TO_GBK[15670] := 16#69CE;
   // UNICODE_TO_GBK[15671] := 16#E9B6;
   // UNICODE_TO_GBK[15672] := 16#69CF;
   // UNICODE_TO_GBK[15673] := 16#988D;
   // UNICODE_TO_GBK[15674] := 16#69D0;
   // UNICODE_TO_GBK[15675] := 16#BBB1;
   // UNICODE_TO_GBK[15676] := 16#69D1;
   // UNICODE_TO_GBK[15677] := 16#988E;
   // UNICODE_TO_GBK[15678] := 16#69D2;
   // UNICODE_TO_GBK[15679] := 16#988F;
   // UNICODE_TO_GBK[15680] := 16#69D3;
   // UNICODE_TO_GBK[15681] := 16#9890;
   // UNICODE_TO_GBK[15682] := 16#69D4;
   // UNICODE_TO_GBK[15683] := 16#E9C0;
   // UNICODE_TO_GBK[15684] := 16#69D5;
   // UNICODE_TO_GBK[15685] := 16#9891;
   // UNICODE_TO_GBK[15686] := 16#69D6;
   // UNICODE_TO_GBK[15687] := 16#9892;
   // UNICODE_TO_GBK[15688] := 16#69D7;
   // UNICODE_TO_GBK[15689] := 16#9893;
   // UNICODE_TO_GBK[15690] := 16#69D8;
   // UNICODE_TO_GBK[15691] := 16#9894;
   // UNICODE_TO_GBK[15692] := 16#69D9;
   // UNICODE_TO_GBK[15693] := 16#9895;
   // UNICODE_TO_GBK[15694] := 16#69DA;
   // UNICODE_TO_GBK[15695] := 16#9896;
   // UNICODE_TO_GBK[15696] := 16#69DB;
   // UNICODE_TO_GBK[15697] := 16#BCF7;
   // UNICODE_TO_GBK[15698] := 16#69DC;
   // UNICODE_TO_GBK[15699] := 16#9897;
   // UNICODE_TO_GBK[15700] := 16#69DD;
   // UNICODE_TO_GBK[15701] := 16#9898;
   // UNICODE_TO_GBK[15702] := 16#69DE;
   // UNICODE_TO_GBK[15703] := 16#9899;
   // UNICODE_TO_GBK[15704] := 16#69DF;
   // UNICODE_TO_GBK[15705] := 16#E9C4;
   // UNICODE_TO_GBK[15706] := 16#69E0;
   // UNICODE_TO_GBK[15707] := 16#E9C6;
   // UNICODE_TO_GBK[15708] := 16#69E1;
   // UNICODE_TO_GBK[15709] := 16#989A;
   // UNICODE_TO_GBK[15710] := 16#69E2;
   // UNICODE_TO_GBK[15711] := 16#989B;
   // UNICODE_TO_GBK[15712] := 16#69E3;
   // UNICODE_TO_GBK[15713] := 16#989C;
   // UNICODE_TO_GBK[15714] := 16#69E4;
   // UNICODE_TO_GBK[15715] := 16#989D;
   // UNICODE_TO_GBK[15716] := 16#69E5;
   // UNICODE_TO_GBK[15717] := 16#989E;
   // UNICODE_TO_GBK[15718] := 16#69E6;
   // UNICODE_TO_GBK[15719] := 16#989F;
   // UNICODE_TO_GBK[15720] := 16#69E7;
   // UNICODE_TO_GBK[15721] := 16#98A0;
   // UNICODE_TO_GBK[15722] := 16#69E8;
   // UNICODE_TO_GBK[15723] := 16#98A1;
   // UNICODE_TO_GBK[15724] := 16#69E9;
   // UNICODE_TO_GBK[15725] := 16#98A2;
   // UNICODE_TO_GBK[15726] := 16#69EA;
   // UNICODE_TO_GBK[15727] := 16#98A3;
   // UNICODE_TO_GBK[15728] := 16#69EB;
   // UNICODE_TO_GBK[15729] := 16#98A4;
   // UNICODE_TO_GBK[15730] := 16#69EC;
   // UNICODE_TO_GBK[15731] := 16#98A5;
   // UNICODE_TO_GBK[15732] := 16#69ED;
   // UNICODE_TO_GBK[15733] := 16#E9CA;
   // UNICODE_TO_GBK[15734] := 16#69EE;
   // UNICODE_TO_GBK[15735] := 16#98A6;
   // UNICODE_TO_GBK[15736] := 16#69EF;
   // UNICODE_TO_GBK[15737] := 16#98A7;
   // UNICODE_TO_GBK[15738] := 16#69F0;
   // UNICODE_TO_GBK[15739] := 16#98A8;
   // UNICODE_TO_GBK[15740] := 16#69F1;
   // UNICODE_TO_GBK[15741] := 16#98A9;
   // UNICODE_TO_GBK[15742] := 16#69F2;
   // UNICODE_TO_GBK[15743] := 16#E9CE;
   // UNICODE_TO_GBK[15744] := 16#69F3;
   // UNICODE_TO_GBK[15745] := 16#98AA;
   // UNICODE_TO_GBK[15746] := 16#69F4;
   // UNICODE_TO_GBK[15747] := 16#98AB;
   // UNICODE_TO_GBK[15748] := 16#69F5;
   // UNICODE_TO_GBK[15749] := 16#98AC;
   // UNICODE_TO_GBK[15750] := 16#69F6;
   // UNICODE_TO_GBK[15751] := 16#98AD;
   // UNICODE_TO_GBK[15752] := 16#69F7;
   // UNICODE_TO_GBK[15753] := 16#98AE;
   // UNICODE_TO_GBK[15754] := 16#69F8;
   // UNICODE_TO_GBK[15755] := 16#98AF;
   // UNICODE_TO_GBK[15756] := 16#69F9;
   // UNICODE_TO_GBK[15757] := 16#98B0;
   // UNICODE_TO_GBK[15758] := 16#69FA;
   // UNICODE_TO_GBK[15759] := 16#98B1;
   // UNICODE_TO_GBK[15760] := 16#69FB;
   // UNICODE_TO_GBK[15761] := 16#98B2;
   // UNICODE_TO_GBK[15762] := 16#69FC;
   // UNICODE_TO_GBK[15763] := 16#98B3;
   // UNICODE_TO_GBK[15764] := 16#69FD;
   // UNICODE_TO_GBK[15765] := 16#B2DB;
   // UNICODE_TO_GBK[15766] := 16#69FE;
   // UNICODE_TO_GBK[15767] := 16#98B4;
   // UNICODE_TO_GBK[15768] := 16#69FF;
   // UNICODE_TO_GBK[15769] := 16#E9C8;
   // UNICODE_TO_GBK[15770] := 16#6A00;
   // UNICODE_TO_GBK[15771] := 16#98B5;
   // UNICODE_TO_GBK[15772] := 16#6A01;
   // UNICODE_TO_GBK[15773] := 16#98B6;
   // UNICODE_TO_GBK[15774] := 16#6A02;
   // UNICODE_TO_GBK[15775] := 16#98B7;
   // UNICODE_TO_GBK[15776] := 16#6A03;
   // UNICODE_TO_GBK[15777] := 16#98B8;
   // UNICODE_TO_GBK[15778] := 16#6A04;
   // UNICODE_TO_GBK[15779] := 16#98B9;
   // UNICODE_TO_GBK[15780] := 16#6A05;
   // UNICODE_TO_GBK[15781] := 16#98BA;
   // UNICODE_TO_GBK[15782] := 16#6A06;
   // UNICODE_TO_GBK[15783] := 16#98BB;
   // UNICODE_TO_GBK[15784] := 16#6A07;
   // UNICODE_TO_GBK[15785] := 16#98BC;
   // UNICODE_TO_GBK[15786] := 16#6A08;
   // UNICODE_TO_GBK[15787] := 16#98BD;
   // UNICODE_TO_GBK[15788] := 16#6A09;
   // UNICODE_TO_GBK[15789] := 16#98BE;
   // UNICODE_TO_GBK[15790] := 16#6A0A;
   // UNICODE_TO_GBK[15791] := 16#B7AE;
   // UNICODE_TO_GBK[15792] := 16#6A0B;
   // UNICODE_TO_GBK[15793] := 16#98BF;
   // UNICODE_TO_GBK[15794] := 16#6A0C;
   // UNICODE_TO_GBK[15795] := 16#98C0;
   // UNICODE_TO_GBK[15796] := 16#6A0D;
   // UNICODE_TO_GBK[15797] := 16#98C1;
   // UNICODE_TO_GBK[15798] := 16#6A0E;
   // UNICODE_TO_GBK[15799] := 16#98C2;
   // UNICODE_TO_GBK[15800] := 16#6A0F;
   // UNICODE_TO_GBK[15801] := 16#98C3;
   // UNICODE_TO_GBK[15802] := 16#6A10;
   // UNICODE_TO_GBK[15803] := 16#98C4;
   // UNICODE_TO_GBK[15804] := 16#6A11;
   // UNICODE_TO_GBK[15805] := 16#98C5;
   // UNICODE_TO_GBK[15806] := 16#6A12;
   // UNICODE_TO_GBK[15807] := 16#98C6;
   // UNICODE_TO_GBK[15808] := 16#6A13;
   // UNICODE_TO_GBK[15809] := 16#98C7;
   // UNICODE_TO_GBK[15810] := 16#6A14;
   // UNICODE_TO_GBK[15811] := 16#98C8;
   // UNICODE_TO_GBK[15812] := 16#6A15;
   // UNICODE_TO_GBK[15813] := 16#98C9;
   // UNICODE_TO_GBK[15814] := 16#6A16;
   // UNICODE_TO_GBK[15815] := 16#98CA;
   // UNICODE_TO_GBK[15816] := 16#6A17;
   // UNICODE_TO_GBK[15817] := 16#E9CB;
   // UNICODE_TO_GBK[15818] := 16#6A18;
   // UNICODE_TO_GBK[15819] := 16#E9CC;
   // UNICODE_TO_GBK[15820] := 16#6A19;
   // UNICODE_TO_GBK[15821] := 16#98CB;
   // UNICODE_TO_GBK[15822] := 16#6A1A;
   // UNICODE_TO_GBK[15823] := 16#98CC;
   // UNICODE_TO_GBK[15824] := 16#6A1B;
   // UNICODE_TO_GBK[15825] := 16#98CD;
   // UNICODE_TO_GBK[15826] := 16#6A1C;
   // UNICODE_TO_GBK[15827] := 16#98CE;
   // UNICODE_TO_GBK[15828] := 16#6A1D;
   // UNICODE_TO_GBK[15829] := 16#98CF;
   // UNICODE_TO_GBK[15830] := 16#6A1E;
   // UNICODE_TO_GBK[15831] := 16#98D0;
   // UNICODE_TO_GBK[15832] := 16#6A1F;
   // UNICODE_TO_GBK[15833] := 16#D5C1;
   // UNICODE_TO_GBK[15834] := 16#6A20;
   // UNICODE_TO_GBK[15835] := 16#98D1;
   // UNICODE_TO_GBK[15836] := 16#6A21;
   // UNICODE_TO_GBK[15837] := 16#C4A3;
   // UNICODE_TO_GBK[15838] := 16#6A22;
   // UNICODE_TO_GBK[15839] := 16#98D2;
   // UNICODE_TO_GBK[15840] := 16#6A23;
   // UNICODE_TO_GBK[15841] := 16#98D3;
   // UNICODE_TO_GBK[15842] := 16#6A24;
   // UNICODE_TO_GBK[15843] := 16#98D4;
   // UNICODE_TO_GBK[15844] := 16#6A25;
   // UNICODE_TO_GBK[15845] := 16#98D5;
   // UNICODE_TO_GBK[15846] := 16#6A26;
   // UNICODE_TO_GBK[15847] := 16#98D6;
   // UNICODE_TO_GBK[15848] := 16#6A27;
   // UNICODE_TO_GBK[15849] := 16#98D7;
   // UNICODE_TO_GBK[15850] := 16#6A28;
   // UNICODE_TO_GBK[15851] := 16#E9D8;
   // UNICODE_TO_GBK[15852] := 16#6A29;
   // UNICODE_TO_GBK[15853] := 16#98D8;
   // UNICODE_TO_GBK[15854] := 16#6A2A;
   // UNICODE_TO_GBK[15855] := 16#BAE1;
   // UNICODE_TO_GBK[15856] := 16#6A2B;
   // UNICODE_TO_GBK[15857] := 16#98D9;
   // UNICODE_TO_GBK[15858] := 16#6A2C;
   // UNICODE_TO_GBK[15859] := 16#98DA;
   // UNICODE_TO_GBK[15860] := 16#6A2D;
   // UNICODE_TO_GBK[15861] := 16#98DB;
   // UNICODE_TO_GBK[15862] := 16#6A2E;
   // UNICODE_TO_GBK[15863] := 16#98DC;
   // UNICODE_TO_GBK[15864] := 16#6A2F;
   // UNICODE_TO_GBK[15865] := 16#E9C9;
   // UNICODE_TO_GBK[15866] := 16#6A30;
   // UNICODE_TO_GBK[15867] := 16#98DD;
   // UNICODE_TO_GBK[15868] := 16#6A31;
   // UNICODE_TO_GBK[15869] := 16#D3A3;
   // UNICODE_TO_GBK[15870] := 16#6A32;
   // UNICODE_TO_GBK[15871] := 16#98DE;
   // UNICODE_TO_GBK[15872] := 16#6A33;
   // UNICODE_TO_GBK[15873] := 16#98DF;
   // UNICODE_TO_GBK[15874] := 16#6A34;
   // UNICODE_TO_GBK[15875] := 16#98E0;
   // UNICODE_TO_GBK[15876] := 16#6A35;
   // UNICODE_TO_GBK[15877] := 16#E9D4;
   // UNICODE_TO_GBK[15878] := 16#6A36;
   // UNICODE_TO_GBK[15879] := 16#98E1;
   // UNICODE_TO_GBK[15880] := 16#6A37;
   // UNICODE_TO_GBK[15881] := 16#98E2;
   // UNICODE_TO_GBK[15882] := 16#6A38;
   // UNICODE_TO_GBK[15883] := 16#98E3;
   // UNICODE_TO_GBK[15884] := 16#6A39;
   // UNICODE_TO_GBK[15885] := 16#98E4;
   // UNICODE_TO_GBK[15886] := 16#6A3A;
   // UNICODE_TO_GBK[15887] := 16#98E5;
   // UNICODE_TO_GBK[15888] := 16#6A3B;
   // UNICODE_TO_GBK[15889] := 16#98E6;
   // UNICODE_TO_GBK[15890] := 16#6A3C;
   // UNICODE_TO_GBK[15891] := 16#98E7;
   // UNICODE_TO_GBK[15892] := 16#6A3D;
   // UNICODE_TO_GBK[15893] := 16#E9D7;
   // UNICODE_TO_GBK[15894] := 16#6A3E;
   // UNICODE_TO_GBK[15895] := 16#E9D0;
   // UNICODE_TO_GBK[15896] := 16#6A3F;
   // UNICODE_TO_GBK[15897] := 16#98E8;
   // UNICODE_TO_GBK[15898] := 16#6A40;
   // UNICODE_TO_GBK[15899] := 16#98E9;
   // UNICODE_TO_GBK[15900] := 16#6A41;
   // UNICODE_TO_GBK[15901] := 16#98EA;
   // UNICODE_TO_GBK[15902] := 16#6A42;
   // UNICODE_TO_GBK[15903] := 16#98EB;
   // UNICODE_TO_GBK[15904] := 16#6A43;
   // UNICODE_TO_GBK[15905] := 16#98EC;
   // UNICODE_TO_GBK[15906] := 16#6A44;
   // UNICODE_TO_GBK[15907] := 16#E9CF;
   // UNICODE_TO_GBK[15908] := 16#6A45;
   // UNICODE_TO_GBK[15909] := 16#98ED;
   // UNICODE_TO_GBK[15910] := 16#6A46;
   // UNICODE_TO_GBK[15911] := 16#98EE;
   // UNICODE_TO_GBK[15912] := 16#6A47;
   // UNICODE_TO_GBK[15913] := 16#C7C1;
   // UNICODE_TO_GBK[15914] := 16#6A48;
   // UNICODE_TO_GBK[15915] := 16#98EF;
   // UNICODE_TO_GBK[15916] := 16#6A49;
   // UNICODE_TO_GBK[15917] := 16#98F0;
   // UNICODE_TO_GBK[15918] := 16#6A4A;
   // UNICODE_TO_GBK[15919] := 16#98F1;
   // UNICODE_TO_GBK[15920] := 16#6A4B;
   // UNICODE_TO_GBK[15921] := 16#98F2;
   // UNICODE_TO_GBK[15922] := 16#6A4C;
   // UNICODE_TO_GBK[15923] := 16#98F3;
   // UNICODE_TO_GBK[15924] := 16#6A4D;
   // UNICODE_TO_GBK[15925] := 16#98F4;
   // UNICODE_TO_GBK[15926] := 16#6A4E;
   // UNICODE_TO_GBK[15927] := 16#98F5;
   // UNICODE_TO_GBK[15928] := 16#6A4F;
   // UNICODE_TO_GBK[15929] := 16#98F6;
   // UNICODE_TO_GBK[15930] := 16#6A50;
   // UNICODE_TO_GBK[15931] := 16#E9D2;
   // UNICODE_TO_GBK[15932] := 16#6A51;
   // UNICODE_TO_GBK[15933] := 16#98F7;
   // UNICODE_TO_GBK[15934] := 16#6A52;
   // UNICODE_TO_GBK[15935] := 16#98F8;
   // UNICODE_TO_GBK[15936] := 16#6A53;
   // UNICODE_TO_GBK[15937] := 16#98F9;
   // UNICODE_TO_GBK[15938] := 16#6A54;
   // UNICODE_TO_GBK[15939] := 16#98FA;
   // UNICODE_TO_GBK[15940] := 16#6A55;
   // UNICODE_TO_GBK[15941] := 16#98FB;
   // UNICODE_TO_GBK[15942] := 16#6A56;
   // UNICODE_TO_GBK[15943] := 16#98FC;
   // UNICODE_TO_GBK[15944] := 16#6A57;
   // UNICODE_TO_GBK[15945] := 16#98FD;
   // UNICODE_TO_GBK[15946] := 16#6A58;
   // UNICODE_TO_GBK[15947] := 16#E9D9;
   // UNICODE_TO_GBK[15948] := 16#6A59;
   // UNICODE_TO_GBK[15949] := 16#B3C8;
   // UNICODE_TO_GBK[15950] := 16#6A5A;
   // UNICODE_TO_GBK[15951] := 16#98FE;
   // UNICODE_TO_GBK[15952] := 16#6A5B;
   // UNICODE_TO_GBK[15953] := 16#E9D3;
   // UNICODE_TO_GBK[15954] := 16#6A5C;
   // UNICODE_TO_GBK[15955] := 16#9940;
   // UNICODE_TO_GBK[15956] := 16#6A5D;
   // UNICODE_TO_GBK[15957] := 16#9941;
   // UNICODE_TO_GBK[15958] := 16#6A5E;
   // UNICODE_TO_GBK[15959] := 16#9942;
   // UNICODE_TO_GBK[15960] := 16#6A5F;
   // UNICODE_TO_GBK[15961] := 16#9943;
   // UNICODE_TO_GBK[15962] := 16#6A60;
   // UNICODE_TO_GBK[15963] := 16#9944;
   // UNICODE_TO_GBK[15964] := 16#6A61;
   // UNICODE_TO_GBK[15965] := 16#CFF0;
   // UNICODE_TO_GBK[15966] := 16#6A62;
   // UNICODE_TO_GBK[15967] := 16#9945;
   // UNICODE_TO_GBK[15968] := 16#6A63;
   // UNICODE_TO_GBK[15969] := 16#9946;
   // UNICODE_TO_GBK[15970] := 16#6A64;
   // UNICODE_TO_GBK[15971] := 16#9947;
   // UNICODE_TO_GBK[15972] := 16#6A65;
   // UNICODE_TO_GBK[15973] := 16#E9CD;
   // UNICODE_TO_GBK[15974] := 16#6A66;
   // UNICODE_TO_GBK[15975] := 16#9948;
   // UNICODE_TO_GBK[15976] := 16#6A67;
   // UNICODE_TO_GBK[15977] := 16#9949;
   // UNICODE_TO_GBK[15978] := 16#6A68;
   // UNICODE_TO_GBK[15979] := 16#994A;
   // UNICODE_TO_GBK[15980] := 16#6A69;
   // UNICODE_TO_GBK[15981] := 16#994B;
   // UNICODE_TO_GBK[15982] := 16#6A6A;
   // UNICODE_TO_GBK[15983] := 16#994C;
   // UNICODE_TO_GBK[15984] := 16#6A6B;
   // UNICODE_TO_GBK[15985] := 16#994D;
   // UNICODE_TO_GBK[15986] := 16#6A6C;
   // UNICODE_TO_GBK[15987] := 16#994E;
   // UNICODE_TO_GBK[15988] := 16#6A6D;
   // UNICODE_TO_GBK[15989] := 16#994F;
   // UNICODE_TO_GBK[15990] := 16#6A6E;
   // UNICODE_TO_GBK[15991] := 16#9950;
   // UNICODE_TO_GBK[15992] := 16#6A6F;
   // UNICODE_TO_GBK[15993] := 16#9951;
   // UNICODE_TO_GBK[15994] := 16#6A70;
   // UNICODE_TO_GBK[15995] := 16#9952;
   // UNICODE_TO_GBK[15996] := 16#6A71;
   // UNICODE_TO_GBK[15997] := 16#B3F7;
   // UNICODE_TO_GBK[15998] := 16#6A72;
   // UNICODE_TO_GBK[15999] := 16#9953;
   // UNICODE_TO_GBK[16000] := 16#6A73;
   // UNICODE_TO_GBK[16001] := 16#9954;
   // UNICODE_TO_GBK[16002] := 16#6A74;
   // UNICODE_TO_GBK[16003] := 16#9955;
   // UNICODE_TO_GBK[16004] := 16#6A75;
   // UNICODE_TO_GBK[16005] := 16#9956;
   // UNICODE_TO_GBK[16006] := 16#6A76;
   // UNICODE_TO_GBK[16007] := 16#9957;
   // UNICODE_TO_GBK[16008] := 16#6A77;
   // UNICODE_TO_GBK[16009] := 16#9958;
   // UNICODE_TO_GBK[16010] := 16#6A78;
   // UNICODE_TO_GBK[16011] := 16#9959;
   // UNICODE_TO_GBK[16012] := 16#6A79;
   // UNICODE_TO_GBK[16013] := 16#E9D6;
   // UNICODE_TO_GBK[16014] := 16#6A7A;
   // UNICODE_TO_GBK[16015] := 16#995A;
   // UNICODE_TO_GBK[16016] := 16#6A7B;
   // UNICODE_TO_GBK[16017] := 16#995B;
   // UNICODE_TO_GBK[16018] := 16#6A7C;
   // UNICODE_TO_GBK[16019] := 16#E9DA;
   // UNICODE_TO_GBK[16020] := 16#6A7D;
   // UNICODE_TO_GBK[16021] := 16#995C;
   // UNICODE_TO_GBK[16022] := 16#6A7E;
   // UNICODE_TO_GBK[16023] := 16#995D;
   // UNICODE_TO_GBK[16024] := 16#6A7F;
   // UNICODE_TO_GBK[16025] := 16#995E;
   // UNICODE_TO_GBK[16026] := 16#6A80;
   // UNICODE_TO_GBK[16027] := 16#CCB4;
   // UNICODE_TO_GBK[16028] := 16#6A81;
   // UNICODE_TO_GBK[16029] := 16#995F;
   // UNICODE_TO_GBK[16030] := 16#6A82;
   // UNICODE_TO_GBK[16031] := 16#9960;
   // UNICODE_TO_GBK[16032] := 16#6A83;
   // UNICODE_TO_GBK[16033] := 16#9961;
   // UNICODE_TO_GBK[16034] := 16#6A84;
   // UNICODE_TO_GBK[16035] := 16#CFAD;
   // UNICODE_TO_GBK[16036] := 16#6A85;
   // UNICODE_TO_GBK[16037] := 16#9962;
   // UNICODE_TO_GBK[16038] := 16#6A86;
   // UNICODE_TO_GBK[16039] := 16#9963;
   // UNICODE_TO_GBK[16040] := 16#6A87;
   // UNICODE_TO_GBK[16041] := 16#9964;
   // UNICODE_TO_GBK[16042] := 16#6A88;
   // UNICODE_TO_GBK[16043] := 16#9965;
   // UNICODE_TO_GBK[16044] := 16#6A89;
   // UNICODE_TO_GBK[16045] := 16#9966;
   // UNICODE_TO_GBK[16046] := 16#6A8A;
   // UNICODE_TO_GBK[16047] := 16#9967;
   // UNICODE_TO_GBK[16048] := 16#6A8B;
   // UNICODE_TO_GBK[16049] := 16#9968;
   // UNICODE_TO_GBK[16050] := 16#6A8C;
   // UNICODE_TO_GBK[16051] := 16#9969;
   // UNICODE_TO_GBK[16052] := 16#6A8D;
   // UNICODE_TO_GBK[16053] := 16#996A;
   // UNICODE_TO_GBK[16054] := 16#6A8E;
   // UNICODE_TO_GBK[16055] := 16#E9D5;
   // UNICODE_TO_GBK[16056] := 16#6A8F;
   // UNICODE_TO_GBK[16057] := 16#996B;
   // UNICODE_TO_GBK[16058] := 16#6A90;
   // UNICODE_TO_GBK[16059] := 16#E9DC;
   // UNICODE_TO_GBK[16060] := 16#6A91;
   // UNICODE_TO_GBK[16061] := 16#E9DB;
   // UNICODE_TO_GBK[16062] := 16#6A92;
   // UNICODE_TO_GBK[16063] := 16#996C;
   // UNICODE_TO_GBK[16064] := 16#6A93;
   // UNICODE_TO_GBK[16065] := 16#996D;
   // UNICODE_TO_GBK[16066] := 16#6A94;
   // UNICODE_TO_GBK[16067] := 16#996E;
   // UNICODE_TO_GBK[16068] := 16#6A95;
   // UNICODE_TO_GBK[16069] := 16#996F;
   // UNICODE_TO_GBK[16070] := 16#6A96;
   // UNICODE_TO_GBK[16071] := 16#9970;
   // UNICODE_TO_GBK[16072] := 16#6A97;
   // UNICODE_TO_GBK[16073] := 16#E9DE;
   // UNICODE_TO_GBK[16074] := 16#6A98;
   // UNICODE_TO_GBK[16075] := 16#9971;
   // UNICODE_TO_GBK[16076] := 16#6A99;
   // UNICODE_TO_GBK[16077] := 16#9972;
   // UNICODE_TO_GBK[16078] := 16#6A9A;
   // UNICODE_TO_GBK[16079] := 16#9973;
   // UNICODE_TO_GBK[16080] := 16#6A9B;
   // UNICODE_TO_GBK[16081] := 16#9974;
   // UNICODE_TO_GBK[16082] := 16#6A9C;
   // UNICODE_TO_GBK[16083] := 16#9975;
   // UNICODE_TO_GBK[16084] := 16#6A9D;
   // UNICODE_TO_GBK[16085] := 16#9976;
   // UNICODE_TO_GBK[16086] := 16#6A9E;
   // UNICODE_TO_GBK[16087] := 16#9977;
   // UNICODE_TO_GBK[16088] := 16#6A9F;
   // UNICODE_TO_GBK[16089] := 16#9978;
   // UNICODE_TO_GBK[16090] := 16#6AA0;
   // UNICODE_TO_GBK[16091] := 16#E9D1;
   // UNICODE_TO_GBK[16092] := 16#6AA1;
   // UNICODE_TO_GBK[16093] := 16#9979;
   // UNICODE_TO_GBK[16094] := 16#6AA2;
   // UNICODE_TO_GBK[16095] := 16#997A;
   // UNICODE_TO_GBK[16096] := 16#6AA3;
   // UNICODE_TO_GBK[16097] := 16#997B;
   // UNICODE_TO_GBK[16098] := 16#6AA4;
   // UNICODE_TO_GBK[16099] := 16#997C;
   // UNICODE_TO_GBK[16100] := 16#6AA5;
   // UNICODE_TO_GBK[16101] := 16#997D;
   // UNICODE_TO_GBK[16102] := 16#6AA6;
   // UNICODE_TO_GBK[16103] := 16#997E;
   // UNICODE_TO_GBK[16104] := 16#6AA7;
   // UNICODE_TO_GBK[16105] := 16#9980;
   // UNICODE_TO_GBK[16106] := 16#6AA8;
   // UNICODE_TO_GBK[16107] := 16#9981;
   // UNICODE_TO_GBK[16108] := 16#6AA9;
   // UNICODE_TO_GBK[16109] := 16#E9DD;
   // UNICODE_TO_GBK[16110] := 16#6AAA;
   // UNICODE_TO_GBK[16111] := 16#9982;
   // UNICODE_TO_GBK[16112] := 16#6AAB;
   // UNICODE_TO_GBK[16113] := 16#E9DF;
   // UNICODE_TO_GBK[16114] := 16#6AAC;
   // UNICODE_TO_GBK[16115] := 16#C3CA;
   // UNICODE_TO_GBK[16116] := 16#6AAD;
   // UNICODE_TO_GBK[16117] := 16#9983;
   // UNICODE_TO_GBK[16118] := 16#6AAE;
   // UNICODE_TO_GBK[16119] := 16#9984;
   // UNICODE_TO_GBK[16120] := 16#6AAF;
   // UNICODE_TO_GBK[16121] := 16#9985;
   // UNICODE_TO_GBK[16122] := 16#6AB0;
   // UNICODE_TO_GBK[16123] := 16#9986;
   // UNICODE_TO_GBK[16124] := 16#6AB1;
   // UNICODE_TO_GBK[16125] := 16#9987;
   // UNICODE_TO_GBK[16126] := 16#6AB2;
   // UNICODE_TO_GBK[16127] := 16#9988;
   // UNICODE_TO_GBK[16128] := 16#6AB3;
   // UNICODE_TO_GBK[16129] := 16#9989;
   // UNICODE_TO_GBK[16130] := 16#6AB4;
   // UNICODE_TO_GBK[16131] := 16#998A;
   // UNICODE_TO_GBK[16132] := 16#6AB5;
   // UNICODE_TO_GBK[16133] := 16#998B;
   // UNICODE_TO_GBK[16134] := 16#6AB6;
   // UNICODE_TO_GBK[16135] := 16#998C;
   // UNICODE_TO_GBK[16136] := 16#6AB7;
   // UNICODE_TO_GBK[16137] := 16#998D;
   // UNICODE_TO_GBK[16138] := 16#6AB8;
   // UNICODE_TO_GBK[16139] := 16#998E;
   // UNICODE_TO_GBK[16140] := 16#6AB9;
   // UNICODE_TO_GBK[16141] := 16#998F;
   // UNICODE_TO_GBK[16142] := 16#6ABA;
   // UNICODE_TO_GBK[16143] := 16#9990;
   // UNICODE_TO_GBK[16144] := 16#6ABB;
   // UNICODE_TO_GBK[16145] := 16#9991;
   // UNICODE_TO_GBK[16146] := 16#6ABC;
   // UNICODE_TO_GBK[16147] := 16#9992;
   // UNICODE_TO_GBK[16148] := 16#6ABD;
   // UNICODE_TO_GBK[16149] := 16#9993;
   // UNICODE_TO_GBK[16150] := 16#6ABE;
   // UNICODE_TO_GBK[16151] := 16#9994;
   // UNICODE_TO_GBK[16152] := 16#6ABF;
   // UNICODE_TO_GBK[16153] := 16#9995;
   // UNICODE_TO_GBK[16154] := 16#6AC0;
   // UNICODE_TO_GBK[16155] := 16#9996;
   // UNICODE_TO_GBK[16156] := 16#6AC1;
   // UNICODE_TO_GBK[16157] := 16#9997;
   // UNICODE_TO_GBK[16158] := 16#6AC2;
   // UNICODE_TO_GBK[16159] := 16#9998;
   // UNICODE_TO_GBK[16160] := 16#6AC3;
   // UNICODE_TO_GBK[16161] := 16#9999;
   // UNICODE_TO_GBK[16162] := 16#6AC4;
   // UNICODE_TO_GBK[16163] := 16#999A;
   // UNICODE_TO_GBK[16164] := 16#6AC5;
   // UNICODE_TO_GBK[16165] := 16#999B;
   // UNICODE_TO_GBK[16166] := 16#6AC6;
   // UNICODE_TO_GBK[16167] := 16#999C;
   // UNICODE_TO_GBK[16168] := 16#6AC7;
   // UNICODE_TO_GBK[16169] := 16#999D;
   // UNICODE_TO_GBK[16170] := 16#6AC8;
   // UNICODE_TO_GBK[16171] := 16#999E;
   // UNICODE_TO_GBK[16172] := 16#6AC9;
   // UNICODE_TO_GBK[16173] := 16#999F;
   // UNICODE_TO_GBK[16174] := 16#6ACA;
   // UNICODE_TO_GBK[16175] := 16#99A0;
   // UNICODE_TO_GBK[16176] := 16#6ACB;
   // UNICODE_TO_GBK[16177] := 16#99A1;
   // UNICODE_TO_GBK[16178] := 16#6ACC;
   // UNICODE_TO_GBK[16179] := 16#99A2;
   // UNICODE_TO_GBK[16180] := 16#6ACD;
   // UNICODE_TO_GBK[16181] := 16#99A3;
   // UNICODE_TO_GBK[16182] := 16#6ACE;
   // UNICODE_TO_GBK[16183] := 16#99A4;
   // UNICODE_TO_GBK[16184] := 16#6ACF;
   // UNICODE_TO_GBK[16185] := 16#99A5;
   // UNICODE_TO_GBK[16186] := 16#6AD0;
   // UNICODE_TO_GBK[16187] := 16#99A6;
   // UNICODE_TO_GBK[16188] := 16#6AD1;
   // UNICODE_TO_GBK[16189] := 16#99A7;
   // UNICODE_TO_GBK[16190] := 16#6AD2;
   // UNICODE_TO_GBK[16191] := 16#99A8;
   // UNICODE_TO_GBK[16192] := 16#6AD3;
   // UNICODE_TO_GBK[16193] := 16#99A9;
   // UNICODE_TO_GBK[16194] := 16#6AD4;
   // UNICODE_TO_GBK[16195] := 16#99AA;
   // UNICODE_TO_GBK[16196] := 16#6AD5;
   // UNICODE_TO_GBK[16197] := 16#99AB;
   // UNICODE_TO_GBK[16198] := 16#6AD6;
   // UNICODE_TO_GBK[16199] := 16#99AC;
   // UNICODE_TO_GBK[16200] := 16#6AD7;
   // UNICODE_TO_GBK[16201] := 16#99AD;
   // UNICODE_TO_GBK[16202] := 16#6AD8;
   // UNICODE_TO_GBK[16203] := 16#99AE;
   // UNICODE_TO_GBK[16204] := 16#6AD9;
   // UNICODE_TO_GBK[16205] := 16#99AF;
   // UNICODE_TO_GBK[16206] := 16#6ADA;
   // UNICODE_TO_GBK[16207] := 16#99B0;
   // UNICODE_TO_GBK[16208] := 16#6ADB;
   // UNICODE_TO_GBK[16209] := 16#99B1;
   // UNICODE_TO_GBK[16210] := 16#6ADC;
   // UNICODE_TO_GBK[16211] := 16#99B2;
   // UNICODE_TO_GBK[16212] := 16#6ADD;
   // UNICODE_TO_GBK[16213] := 16#99B3;
   // UNICODE_TO_GBK[16214] := 16#6ADE;
   // UNICODE_TO_GBK[16215] := 16#99B4;
   // UNICODE_TO_GBK[16216] := 16#6ADF;
   // UNICODE_TO_GBK[16217] := 16#99B5;
   // UNICODE_TO_GBK[16218] := 16#6AE0;
   // UNICODE_TO_GBK[16219] := 16#99B6;
   // UNICODE_TO_GBK[16220] := 16#6AE1;
   // UNICODE_TO_GBK[16221] := 16#99B7;
   // UNICODE_TO_GBK[16222] := 16#6AE2;
   // UNICODE_TO_GBK[16223] := 16#99B8;
   // UNICODE_TO_GBK[16224] := 16#6AE3;
   // UNICODE_TO_GBK[16225] := 16#99B9;
   // UNICODE_TO_GBK[16226] := 16#6AE4;
   // UNICODE_TO_GBK[16227] := 16#99BA;
   // UNICODE_TO_GBK[16228] := 16#6AE5;
   // UNICODE_TO_GBK[16229] := 16#99BB;
   // UNICODE_TO_GBK[16230] := 16#6AE6;
   // UNICODE_TO_GBK[16231] := 16#99BC;
   // UNICODE_TO_GBK[16232] := 16#6AE7;
   // UNICODE_TO_GBK[16233] := 16#99BD;
   // UNICODE_TO_GBK[16234] := 16#6AE8;
   // UNICODE_TO_GBK[16235] := 16#99BE;
   // UNICODE_TO_GBK[16236] := 16#6AE9;
   // UNICODE_TO_GBK[16237] := 16#99BF;
   // UNICODE_TO_GBK[16238] := 16#6AEA;
   // UNICODE_TO_GBK[16239] := 16#99C0;
   // UNICODE_TO_GBK[16240] := 16#6AEB;
   // UNICODE_TO_GBK[16241] := 16#99C1;
   // UNICODE_TO_GBK[16242] := 16#6AEC;
   // UNICODE_TO_GBK[16243] := 16#99C2;
   // UNICODE_TO_GBK[16244] := 16#6AED;
   // UNICODE_TO_GBK[16245] := 16#99C3;
   // UNICODE_TO_GBK[16246] := 16#6AEE;
   // UNICODE_TO_GBK[16247] := 16#99C4;
   // UNICODE_TO_GBK[16248] := 16#6AEF;
   // UNICODE_TO_GBK[16249] := 16#99C5;
   // UNICODE_TO_GBK[16250] := 16#6AF0;
   // UNICODE_TO_GBK[16251] := 16#99C6;
   // UNICODE_TO_GBK[16252] := 16#6AF1;
   // UNICODE_TO_GBK[16253] := 16#99C7;
   // UNICODE_TO_GBK[16254] := 16#6AF2;
   // UNICODE_TO_GBK[16255] := 16#99C8;
   // UNICODE_TO_GBK[16256] := 16#6AF3;
   // UNICODE_TO_GBK[16257] := 16#99C9;
   // UNICODE_TO_GBK[16258] := 16#6AF4;
   // UNICODE_TO_GBK[16259] := 16#99CA;
   // UNICODE_TO_GBK[16260] := 16#6AF5;
   // UNICODE_TO_GBK[16261] := 16#99CB;
   // UNICODE_TO_GBK[16262] := 16#6AF6;
   // UNICODE_TO_GBK[16263] := 16#99CC;
   // UNICODE_TO_GBK[16264] := 16#6AF7;
   // UNICODE_TO_GBK[16265] := 16#99CD;
   // UNICODE_TO_GBK[16266] := 16#6AF8;
   // UNICODE_TO_GBK[16267] := 16#99CE;
   // UNICODE_TO_GBK[16268] := 16#6AF9;
   // UNICODE_TO_GBK[16269] := 16#99CF;
   // UNICODE_TO_GBK[16270] := 16#6AFA;
   // UNICODE_TO_GBK[16271] := 16#99D0;
   // UNICODE_TO_GBK[16272] := 16#6AFB;
   // UNICODE_TO_GBK[16273] := 16#99D1;
   // UNICODE_TO_GBK[16274] := 16#6AFC;
   // UNICODE_TO_GBK[16275] := 16#99D2;
   // UNICODE_TO_GBK[16276] := 16#6AFD;
   // UNICODE_TO_GBK[16277] := 16#99D3;
   // UNICODE_TO_GBK[16278] := 16#6AFE;
   // UNICODE_TO_GBK[16279] := 16#99D4;
   // UNICODE_TO_GBK[16280] := 16#6AFF;
   // UNICODE_TO_GBK[16281] := 16#99D5;
   // UNICODE_TO_GBK[16282] := 16#6B00;
   // UNICODE_TO_GBK[16283] := 16#99D6;
   // UNICODE_TO_GBK[16284] := 16#6B01;
   // UNICODE_TO_GBK[16285] := 16#99D7;
   // UNICODE_TO_GBK[16286] := 16#6B02;
   // UNICODE_TO_GBK[16287] := 16#99D8;
   // UNICODE_TO_GBK[16288] := 16#6B03;
   // UNICODE_TO_GBK[16289] := 16#99D9;
   // UNICODE_TO_GBK[16290] := 16#6B04;
   // UNICODE_TO_GBK[16291] := 16#99DA;
   // UNICODE_TO_GBK[16292] := 16#6B05;
   // UNICODE_TO_GBK[16293] := 16#99DB;
   // UNICODE_TO_GBK[16294] := 16#6B06;
   // UNICODE_TO_GBK[16295] := 16#99DC;
   // UNICODE_TO_GBK[16296] := 16#6B07;
   // UNICODE_TO_GBK[16297] := 16#99DD;
   // UNICODE_TO_GBK[16298] := 16#6B08;
   // UNICODE_TO_GBK[16299] := 16#99DE;
   // UNICODE_TO_GBK[16300] := 16#6B09;
   // UNICODE_TO_GBK[16301] := 16#99DF;
   // UNICODE_TO_GBK[16302] := 16#6B0A;
   // UNICODE_TO_GBK[16303] := 16#99E0;
   // UNICODE_TO_GBK[16304] := 16#6B0B;
   // UNICODE_TO_GBK[16305] := 16#99E1;
   // UNICODE_TO_GBK[16306] := 16#6B0C;
   // UNICODE_TO_GBK[16307] := 16#99E2;
   // UNICODE_TO_GBK[16308] := 16#6B0D;
   // UNICODE_TO_GBK[16309] := 16#99E3;
   // UNICODE_TO_GBK[16310] := 16#6B0E;
   // UNICODE_TO_GBK[16311] := 16#99E4;
   // UNICODE_TO_GBK[16312] := 16#6B0F;
   // UNICODE_TO_GBK[16313] := 16#99E5;
   // UNICODE_TO_GBK[16314] := 16#6B10;
   // UNICODE_TO_GBK[16315] := 16#99E6;
   // UNICODE_TO_GBK[16316] := 16#6B11;
   // UNICODE_TO_GBK[16317] := 16#99E7;
   // UNICODE_TO_GBK[16318] := 16#6B12;
   // UNICODE_TO_GBK[16319] := 16#99E8;
   // UNICODE_TO_GBK[16320] := 16#6B13;
   // UNICODE_TO_GBK[16321] := 16#99E9;
   // UNICODE_TO_GBK[16322] := 16#6B14;
   // UNICODE_TO_GBK[16323] := 16#99EA;
   // UNICODE_TO_GBK[16324] := 16#6B15;
   // UNICODE_TO_GBK[16325] := 16#99EB;
   // UNICODE_TO_GBK[16326] := 16#6B16;
   // UNICODE_TO_GBK[16327] := 16#99EC;
   // UNICODE_TO_GBK[16328] := 16#6B17;
   // UNICODE_TO_GBK[16329] := 16#99ED;
   // UNICODE_TO_GBK[16330] := 16#6B18;
   // UNICODE_TO_GBK[16331] := 16#99EE;
   // UNICODE_TO_GBK[16332] := 16#6B19;
   // UNICODE_TO_GBK[16333] := 16#99EF;
   // UNICODE_TO_GBK[16334] := 16#6B1A;
   // UNICODE_TO_GBK[16335] := 16#99F0;
   // UNICODE_TO_GBK[16336] := 16#6B1B;
   // UNICODE_TO_GBK[16337] := 16#99F1;
   // UNICODE_TO_GBK[16338] := 16#6B1C;
   // UNICODE_TO_GBK[16339] := 16#99F2;
   // UNICODE_TO_GBK[16340] := 16#6B1D;
   // UNICODE_TO_GBK[16341] := 16#99F3;
   // UNICODE_TO_GBK[16342] := 16#6B1E;
   // UNICODE_TO_GBK[16343] := 16#99F4;
   // UNICODE_TO_GBK[16344] := 16#6B1F;
   // UNICODE_TO_GBK[16345] := 16#99F5;
   // UNICODE_TO_GBK[16346] := 16#6B20;
   // UNICODE_TO_GBK[16347] := 16#C7B7;
   // UNICODE_TO_GBK[16348] := 16#6B21;
   // UNICODE_TO_GBK[16349] := 16#B4CE;
   // UNICODE_TO_GBK[16350] := 16#6B22;
   // UNICODE_TO_GBK[16351] := 16#BBB6;
   // UNICODE_TO_GBK[16352] := 16#6B23;
   // UNICODE_TO_GBK[16353] := 16#D0C0;
   // UNICODE_TO_GBK[16354] := 16#6B24;
   // UNICODE_TO_GBK[16355] := 16#ECA3;
   // UNICODE_TO_GBK[16356] := 16#6B25;
   // UNICODE_TO_GBK[16357] := 16#99F6;
   // UNICODE_TO_GBK[16358] := 16#6B26;
   // UNICODE_TO_GBK[16359] := 16#99F7;
   // UNICODE_TO_GBK[16360] := 16#6B27;
   // UNICODE_TO_GBK[16361] := 16#C5B7;
   // UNICODE_TO_GBK[16362] := 16#6B28;
   // UNICODE_TO_GBK[16363] := 16#99F8;
   // UNICODE_TO_GBK[16364] := 16#6B29;
   // UNICODE_TO_GBK[16365] := 16#99F9;
   // UNICODE_TO_GBK[16366] := 16#6B2A;
   // UNICODE_TO_GBK[16367] := 16#99FA;
   // UNICODE_TO_GBK[16368] := 16#6B2B;
   // UNICODE_TO_GBK[16369] := 16#99FB;
   // UNICODE_TO_GBK[16370] := 16#6B2C;
   // UNICODE_TO_GBK[16371] := 16#99FC;
   // UNICODE_TO_GBK[16372] := 16#6B2D;
   // UNICODE_TO_GBK[16373] := 16#99FD;
   // UNICODE_TO_GBK[16374] := 16#6B2E;
   // UNICODE_TO_GBK[16375] := 16#99FE;
   // UNICODE_TO_GBK[16376] := 16#6B2F;
   // UNICODE_TO_GBK[16377] := 16#9A40;
   // UNICODE_TO_GBK[16378] := 16#6B30;
   // UNICODE_TO_GBK[16379] := 16#9A41;
   // UNICODE_TO_GBK[16380] := 16#6B31;
   // UNICODE_TO_GBK[16381] := 16#9A42;
   // UNICODE_TO_GBK[16382] := 16#6B32;
   // UNICODE_TO_GBK[16383] := 16#D3FB;
   // UNICODE_TO_GBK[16384] := 16#6B33;
   // UNICODE_TO_GBK[16385] := 16#9A43;
   // UNICODE_TO_GBK[16386] := 16#6B34;
   // UNICODE_TO_GBK[16387] := 16#9A44;
   // UNICODE_TO_GBK[16388] := 16#6B35;
   // UNICODE_TO_GBK[16389] := 16#9A45;
   // UNICODE_TO_GBK[16390] := 16#6B36;
   // UNICODE_TO_GBK[16391] := 16#9A46;
   // UNICODE_TO_GBK[16392] := 16#6B37;
   // UNICODE_TO_GBK[16393] := 16#ECA4;
   // UNICODE_TO_GBK[16394] := 16#6B38;
   // UNICODE_TO_GBK[16395] := 16#9A47;
   // UNICODE_TO_GBK[16396] := 16#6B39;
   // UNICODE_TO_GBK[16397] := 16#ECA5;
   // UNICODE_TO_GBK[16398] := 16#6B3A;
   // UNICODE_TO_GBK[16399] := 16#C6DB;
   // UNICODE_TO_GBK[16400] := 16#6B3B;
   // UNICODE_TO_GBK[16401] := 16#9A48;
   // UNICODE_TO_GBK[16402] := 16#6B3C;
   // UNICODE_TO_GBK[16403] := 16#9A49;
   // UNICODE_TO_GBK[16404] := 16#6B3D;
   // UNICODE_TO_GBK[16405] := 16#9A4A;
   // UNICODE_TO_GBK[16406] := 16#6B3E;
   // UNICODE_TO_GBK[16407] := 16#BFEE;
   // UNICODE_TO_GBK[16408] := 16#6B3F;
   // UNICODE_TO_GBK[16409] := 16#9A4B;
   // UNICODE_TO_GBK[16410] := 16#6B40;
   // UNICODE_TO_GBK[16411] := 16#9A4C;
   // UNICODE_TO_GBK[16412] := 16#6B41;
   // UNICODE_TO_GBK[16413] := 16#9A4D;
   // UNICODE_TO_GBK[16414] := 16#6B42;
   // UNICODE_TO_GBK[16415] := 16#9A4E;
   // UNICODE_TO_GBK[16416] := 16#6B43;
   // UNICODE_TO_GBK[16417] := 16#ECA6;
   // UNICODE_TO_GBK[16418] := 16#6B44;
   // UNICODE_TO_GBK[16419] := 16#9A4F;
   // UNICODE_TO_GBK[16420] := 16#6B45;
   // UNICODE_TO_GBK[16421] := 16#9A50;
   // UNICODE_TO_GBK[16422] := 16#6B46;
   // UNICODE_TO_GBK[16423] := 16#ECA7;
   // UNICODE_TO_GBK[16424] := 16#6B47;
   // UNICODE_TO_GBK[16425] := 16#D0AA;
   // UNICODE_TO_GBK[16426] := 16#6B48;
   // UNICODE_TO_GBK[16427] := 16#9A51;
   // UNICODE_TO_GBK[16428] := 16#6B49;
   // UNICODE_TO_GBK[16429] := 16#C7B8;
   // UNICODE_TO_GBK[16430] := 16#6B4A;
   // UNICODE_TO_GBK[16431] := 16#9A52;
   // UNICODE_TO_GBK[16432] := 16#6B4B;
   // UNICODE_TO_GBK[16433] := 16#9A53;
   // UNICODE_TO_GBK[16434] := 16#6B4C;
   // UNICODE_TO_GBK[16435] := 16#B8E8;
   // UNICODE_TO_GBK[16436] := 16#6B4D;
   // UNICODE_TO_GBK[16437] := 16#9A54;
   // UNICODE_TO_GBK[16438] := 16#6B4E;
   // UNICODE_TO_GBK[16439] := 16#9A55;
   // UNICODE_TO_GBK[16440] := 16#6B4F;
   // UNICODE_TO_GBK[16441] := 16#9A56;
   // UNICODE_TO_GBK[16442] := 16#6B50;
   // UNICODE_TO_GBK[16443] := 16#9A57;
   // UNICODE_TO_GBK[16444] := 16#6B51;
   // UNICODE_TO_GBK[16445] := 16#9A58;
   // UNICODE_TO_GBK[16446] := 16#6B52;
   // UNICODE_TO_GBK[16447] := 16#9A59;
   // UNICODE_TO_GBK[16448] := 16#6B53;
   // UNICODE_TO_GBK[16449] := 16#9A5A;
   // UNICODE_TO_GBK[16450] := 16#6B54;
   // UNICODE_TO_GBK[16451] := 16#9A5B;
   // UNICODE_TO_GBK[16452] := 16#6B55;
   // UNICODE_TO_GBK[16453] := 16#9A5C;
   // UNICODE_TO_GBK[16454] := 16#6B56;
   // UNICODE_TO_GBK[16455] := 16#9A5D;
   // UNICODE_TO_GBK[16456] := 16#6B57;
   // UNICODE_TO_GBK[16457] := 16#9A5E;
   // UNICODE_TO_GBK[16458] := 16#6B58;
   // UNICODE_TO_GBK[16459] := 16#9A5F;
   // UNICODE_TO_GBK[16460] := 16#6B59;
   // UNICODE_TO_GBK[16461] := 16#ECA8;
   // UNICODE_TO_GBK[16462] := 16#6B5A;
   // UNICODE_TO_GBK[16463] := 16#9A60;
   // UNICODE_TO_GBK[16464] := 16#6B5B;
   // UNICODE_TO_GBK[16465] := 16#9A61;
   // UNICODE_TO_GBK[16466] := 16#6B5C;
   // UNICODE_TO_GBK[16467] := 16#9A62;
   // UNICODE_TO_GBK[16468] := 16#6B5D;
   // UNICODE_TO_GBK[16469] := 16#9A63;
   // UNICODE_TO_GBK[16470] := 16#6B5E;
   // UNICODE_TO_GBK[16471] := 16#9A64;
   // UNICODE_TO_GBK[16472] := 16#6B5F;
   // UNICODE_TO_GBK[16473] := 16#9A65;
   // UNICODE_TO_GBK[16474] := 16#6B60;
   // UNICODE_TO_GBK[16475] := 16#9A66;
   // UNICODE_TO_GBK[16476] := 16#6B61;
   // UNICODE_TO_GBK[16477] := 16#9A67;
   // UNICODE_TO_GBK[16478] := 16#6B62;
   // UNICODE_TO_GBK[16479] := 16#D6B9;
   // UNICODE_TO_GBK[16480] := 16#6B63;
   // UNICODE_TO_GBK[16481] := 16#D5FD;
   // UNICODE_TO_GBK[16482] := 16#6B64;
   // UNICODE_TO_GBK[16483] := 16#B4CB;
   // UNICODE_TO_GBK[16484] := 16#6B65;
   // UNICODE_TO_GBK[16485] := 16#B2BD;
   // UNICODE_TO_GBK[16486] := 16#6B66;
   // UNICODE_TO_GBK[16487] := 16#CEE4;
   // UNICODE_TO_GBK[16488] := 16#6B67;
   // UNICODE_TO_GBK[16489] := 16#C6E7;
   // UNICODE_TO_GBK[16490] := 16#6B68;
   // UNICODE_TO_GBK[16491] := 16#9A68;
   // UNICODE_TO_GBK[16492] := 16#6B69;
   // UNICODE_TO_GBK[16493] := 16#9A69;
   // UNICODE_TO_GBK[16494] := 16#6B6A;
   // UNICODE_TO_GBK[16495] := 16#CDE1;
   // UNICODE_TO_GBK[16496] := 16#6B6B;
   // UNICODE_TO_GBK[16497] := 16#9A6A;
   // UNICODE_TO_GBK[16498] := 16#6B6C;
   // UNICODE_TO_GBK[16499] := 16#9A6B;
   // UNICODE_TO_GBK[16500] := 16#6B6D;
   // UNICODE_TO_GBK[16501] := 16#9A6C;
   // UNICODE_TO_GBK[16502] := 16#6B6E;
   // UNICODE_TO_GBK[16503] := 16#9A6D;
   // UNICODE_TO_GBK[16504] := 16#6B6F;
   // UNICODE_TO_GBK[16505] := 16#9A6E;
   // UNICODE_TO_GBK[16506] := 16#6B70;
   // UNICODE_TO_GBK[16507] := 16#9A6F;
   // UNICODE_TO_GBK[16508] := 16#6B71;
   // UNICODE_TO_GBK[16509] := 16#9A70;
   // UNICODE_TO_GBK[16510] := 16#6B72;
   // UNICODE_TO_GBK[16511] := 16#9A71;
   // UNICODE_TO_GBK[16512] := 16#6B73;
   // UNICODE_TO_GBK[16513] := 16#9A72;
   // UNICODE_TO_GBK[16514] := 16#6B74;
   // UNICODE_TO_GBK[16515] := 16#9A73;
   // UNICODE_TO_GBK[16516] := 16#6B75;
   // UNICODE_TO_GBK[16517] := 16#9A74;
   // UNICODE_TO_GBK[16518] := 16#6B76;
   // UNICODE_TO_GBK[16519] := 16#9A75;
   // UNICODE_TO_GBK[16520] := 16#6B77;
   // UNICODE_TO_GBK[16521] := 16#9A76;
   // UNICODE_TO_GBK[16522] := 16#6B78;
   // UNICODE_TO_GBK[16523] := 16#9A77;
   // UNICODE_TO_GBK[16524] := 16#6B79;
   // UNICODE_TO_GBK[16525] := 16#B4F5;
   // UNICODE_TO_GBK[16526] := 16#6B7A;
   // UNICODE_TO_GBK[16527] := 16#9A78;
   // UNICODE_TO_GBK[16528] := 16#6B7B;
   // UNICODE_TO_GBK[16529] := 16#CBC0;
   // UNICODE_TO_GBK[16530] := 16#6B7C;
   // UNICODE_TO_GBK[16531] := 16#BCDF;
   // UNICODE_TO_GBK[16532] := 16#6B7D;
   // UNICODE_TO_GBK[16533] := 16#9A79;
   // UNICODE_TO_GBK[16534] := 16#6B7E;
   // UNICODE_TO_GBK[16535] := 16#9A7A;
   // UNICODE_TO_GBK[16536] := 16#6B7F;
   // UNICODE_TO_GBK[16537] := 16#9A7B;
   // UNICODE_TO_GBK[16538] := 16#6B80;
   // UNICODE_TO_GBK[16539] := 16#9A7C;
   // UNICODE_TO_GBK[16540] := 16#6B81;
   // UNICODE_TO_GBK[16541] := 16#E9E2;
   // UNICODE_TO_GBK[16542] := 16#6B82;
   // UNICODE_TO_GBK[16543] := 16#E9E3;
   // UNICODE_TO_GBK[16544] := 16#6B83;
   // UNICODE_TO_GBK[16545] := 16#D1EA;
   // UNICODE_TO_GBK[16546] := 16#6B84;
   // UNICODE_TO_GBK[16547] := 16#E9E5;
   // UNICODE_TO_GBK[16548] := 16#6B85;
   // UNICODE_TO_GBK[16549] := 16#9A7D;
   // UNICODE_TO_GBK[16550] := 16#6B86;
   // UNICODE_TO_GBK[16551] := 16#B4F9;
   // UNICODE_TO_GBK[16552] := 16#6B87;
   // UNICODE_TO_GBK[16553] := 16#E9E4;
   // UNICODE_TO_GBK[16554] := 16#6B88;
   // UNICODE_TO_GBK[16555] := 16#9A7E;
   // UNICODE_TO_GBK[16556] := 16#6B89;
   // UNICODE_TO_GBK[16557] := 16#D1B3;
   // UNICODE_TO_GBK[16558] := 16#6B8A;
   // UNICODE_TO_GBK[16559] := 16#CAE2;
   // UNICODE_TO_GBK[16560] := 16#6B8B;
   // UNICODE_TO_GBK[16561] := 16#B2D0;
   // UNICODE_TO_GBK[16562] := 16#6B8C;
   // UNICODE_TO_GBK[16563] := 16#9A80;
   // UNICODE_TO_GBK[16564] := 16#6B8D;
   // UNICODE_TO_GBK[16565] := 16#E9E8;
   // UNICODE_TO_GBK[16566] := 16#6B8E;
   // UNICODE_TO_GBK[16567] := 16#9A81;
   // UNICODE_TO_GBK[16568] := 16#6B8F;
   // UNICODE_TO_GBK[16569] := 16#9A82;
   // UNICODE_TO_GBK[16570] := 16#6B90;
   // UNICODE_TO_GBK[16571] := 16#9A83;
   // UNICODE_TO_GBK[16572] := 16#6B91;
   // UNICODE_TO_GBK[16573] := 16#9A84;
   // UNICODE_TO_GBK[16574] := 16#6B92;
   // UNICODE_TO_GBK[16575] := 16#E9E6;
   // UNICODE_TO_GBK[16576] := 16#6B93;
   // UNICODE_TO_GBK[16577] := 16#E9E7;
   // UNICODE_TO_GBK[16578] := 16#6B94;
   // UNICODE_TO_GBK[16579] := 16#9A85;
   // UNICODE_TO_GBK[16580] := 16#6B95;
   // UNICODE_TO_GBK[16581] := 16#9A86;
   // UNICODE_TO_GBK[16582] := 16#6B96;
   // UNICODE_TO_GBK[16583] := 16#D6B3;
   // UNICODE_TO_GBK[16584] := 16#6B97;
   // UNICODE_TO_GBK[16585] := 16#9A87;
   // UNICODE_TO_GBK[16586] := 16#6B98;
   // UNICODE_TO_GBK[16587] := 16#9A88;
   // UNICODE_TO_GBK[16588] := 16#6B99;
   // UNICODE_TO_GBK[16589] := 16#9A89;
   // UNICODE_TO_GBK[16590] := 16#6B9A;
   // UNICODE_TO_GBK[16591] := 16#E9E9;
   // UNICODE_TO_GBK[16592] := 16#6B9B;
   // UNICODE_TO_GBK[16593] := 16#E9EA;
   // UNICODE_TO_GBK[16594] := 16#6B9C;
   // UNICODE_TO_GBK[16595] := 16#9A8A;
   // UNICODE_TO_GBK[16596] := 16#6B9D;
   // UNICODE_TO_GBK[16597] := 16#9A8B;
   // UNICODE_TO_GBK[16598] := 16#6B9E;
   // UNICODE_TO_GBK[16599] := 16#9A8C;
   // UNICODE_TO_GBK[16600] := 16#6B9F;
   // UNICODE_TO_GBK[16601] := 16#9A8D;
   // UNICODE_TO_GBK[16602] := 16#6BA0;
   // UNICODE_TO_GBK[16603] := 16#9A8E;
   // UNICODE_TO_GBK[16604] := 16#6BA1;
   // UNICODE_TO_GBK[16605] := 16#E9EB;
   // UNICODE_TO_GBK[16606] := 16#6BA2;
   // UNICODE_TO_GBK[16607] := 16#9A8F;
   // UNICODE_TO_GBK[16608] := 16#6BA3;
   // UNICODE_TO_GBK[16609] := 16#9A90;
   // UNICODE_TO_GBK[16610] := 16#6BA4;
   // UNICODE_TO_GBK[16611] := 16#9A91;
   // UNICODE_TO_GBK[16612] := 16#6BA5;
   // UNICODE_TO_GBK[16613] := 16#9A92;
   // UNICODE_TO_GBK[16614] := 16#6BA6;
   // UNICODE_TO_GBK[16615] := 16#9A93;
   // UNICODE_TO_GBK[16616] := 16#6BA7;
   // UNICODE_TO_GBK[16617] := 16#9A94;
   // UNICODE_TO_GBK[16618] := 16#6BA8;
   // UNICODE_TO_GBK[16619] := 16#9A95;
   // UNICODE_TO_GBK[16620] := 16#6BA9;
   // UNICODE_TO_GBK[16621] := 16#9A96;
   // UNICODE_TO_GBK[16622] := 16#6BAA;
   // UNICODE_TO_GBK[16623] := 16#E9EC;
   // UNICODE_TO_GBK[16624] := 16#6BAB;
   // UNICODE_TO_GBK[16625] := 16#9A97;
   // UNICODE_TO_GBK[16626] := 16#6BAC;
   // UNICODE_TO_GBK[16627] := 16#9A98;
   // UNICODE_TO_GBK[16628] := 16#6BAD;
   // UNICODE_TO_GBK[16629] := 16#9A99;
   // UNICODE_TO_GBK[16630] := 16#6BAE;
   // UNICODE_TO_GBK[16631] := 16#9A9A;
   // UNICODE_TO_GBK[16632] := 16#6BAF;
   // UNICODE_TO_GBK[16633] := 16#9A9B;
   // UNICODE_TO_GBK[16634] := 16#6BB0;
   // UNICODE_TO_GBK[16635] := 16#9A9C;
   // UNICODE_TO_GBK[16636] := 16#6BB1;
   // UNICODE_TO_GBK[16637] := 16#9A9D;
   // UNICODE_TO_GBK[16638] := 16#6BB2;
   // UNICODE_TO_GBK[16639] := 16#9A9E;
   // UNICODE_TO_GBK[16640] := 16#6BB3;
   // UNICODE_TO_GBK[16641] := 16#ECAF;
   // UNICODE_TO_GBK[16642] := 16#6BB4;
   // UNICODE_TO_GBK[16643] := 16#C5B9;
   // UNICODE_TO_GBK[16644] := 16#6BB5;
   // UNICODE_TO_GBK[16645] := 16#B6CE;
   // UNICODE_TO_GBK[16646] := 16#6BB6;
   // UNICODE_TO_GBK[16647] := 16#9A9F;
   // UNICODE_TO_GBK[16648] := 16#6BB7;
   // UNICODE_TO_GBK[16649] := 16#D2F3;
   // UNICODE_TO_GBK[16650] := 16#6BB8;
   // UNICODE_TO_GBK[16651] := 16#9AA0;
   // UNICODE_TO_GBK[16652] := 16#6BB9;
   // UNICODE_TO_GBK[16653] := 16#9AA1;
   // UNICODE_TO_GBK[16654] := 16#6BBA;
   // UNICODE_TO_GBK[16655] := 16#9AA2;
   // UNICODE_TO_GBK[16656] := 16#6BBB;
   // UNICODE_TO_GBK[16657] := 16#9AA3;
   // UNICODE_TO_GBK[16658] := 16#6BBC;
   // UNICODE_TO_GBK[16659] := 16#9AA4;
   // UNICODE_TO_GBK[16660] := 16#6BBD;
   // UNICODE_TO_GBK[16661] := 16#9AA5;
   // UNICODE_TO_GBK[16662] := 16#6BBE;
   // UNICODE_TO_GBK[16663] := 16#9AA6;
   // UNICODE_TO_GBK[16664] := 16#6BBF;
   // UNICODE_TO_GBK[16665] := 16#B5EE;
   // UNICODE_TO_GBK[16666] := 16#6BC0;
   // UNICODE_TO_GBK[16667] := 16#9AA7;
   // UNICODE_TO_GBK[16668] := 16#6BC1;
   // UNICODE_TO_GBK[16669] := 16#BBD9;
   // UNICODE_TO_GBK[16670] := 16#6BC2;
   // UNICODE_TO_GBK[16671] := 16#ECB1;
   // UNICODE_TO_GBK[16672] := 16#6BC3;
   // UNICODE_TO_GBK[16673] := 16#9AA8;
   // UNICODE_TO_GBK[16674] := 16#6BC4;
   // UNICODE_TO_GBK[16675] := 16#9AA9;
   // UNICODE_TO_GBK[16676] := 16#6BC5;
   // UNICODE_TO_GBK[16677] := 16#D2E3;
   // UNICODE_TO_GBK[16678] := 16#6BC6;
   // UNICODE_TO_GBK[16679] := 16#9AAA;
   // UNICODE_TO_GBK[16680] := 16#6BC7;
   // UNICODE_TO_GBK[16681] := 16#9AAB;
   // UNICODE_TO_GBK[16682] := 16#6BC8;
   // UNICODE_TO_GBK[16683] := 16#9AAC;
   // UNICODE_TO_GBK[16684] := 16#6BC9;
   // UNICODE_TO_GBK[16685] := 16#9AAD;
   // UNICODE_TO_GBK[16686] := 16#6BCA;
   // UNICODE_TO_GBK[16687] := 16#9AAE;
   // UNICODE_TO_GBK[16688] := 16#6BCB;
   // UNICODE_TO_GBK[16689] := 16#CEE3;
   // UNICODE_TO_GBK[16690] := 16#6BCC;
   // UNICODE_TO_GBK[16691] := 16#9AAF;
   // UNICODE_TO_GBK[16692] := 16#6BCD;
   // UNICODE_TO_GBK[16693] := 16#C4B8;
   // UNICODE_TO_GBK[16694] := 16#6BCE;
   // UNICODE_TO_GBK[16695] := 16#9AB0;
   // UNICODE_TO_GBK[16696] := 16#6BCF;
   // UNICODE_TO_GBK[16697] := 16#C3BF;
   // UNICODE_TO_GBK[16698] := 16#6BD0;
   // UNICODE_TO_GBK[16699] := 16#9AB1;
   // UNICODE_TO_GBK[16700] := 16#6BD1;
   // UNICODE_TO_GBK[16701] := 16#9AB2;
   // UNICODE_TO_GBK[16702] := 16#6BD2;
   // UNICODE_TO_GBK[16703] := 16#B6BE;
   // UNICODE_TO_GBK[16704] := 16#6BD3;
   // UNICODE_TO_GBK[16705] := 16#D8B9;
   // UNICODE_TO_GBK[16706] := 16#6BD4;
   // UNICODE_TO_GBK[16707] := 16#B1C8;
   // UNICODE_TO_GBK[16708] := 16#6BD5;
   // UNICODE_TO_GBK[16709] := 16#B1CF;
   // UNICODE_TO_GBK[16710] := 16#6BD6;
   // UNICODE_TO_GBK[16711] := 16#B1D1;
   // UNICODE_TO_GBK[16712] := 16#6BD7;
   // UNICODE_TO_GBK[16713] := 16#C5FE;
   // UNICODE_TO_GBK[16714] := 16#6BD8;
   // UNICODE_TO_GBK[16715] := 16#9AB3;
   // UNICODE_TO_GBK[16716] := 16#6BD9;
   // UNICODE_TO_GBK[16717] := 16#B1D0;
   // UNICODE_TO_GBK[16718] := 16#6BDA;
   // UNICODE_TO_GBK[16719] := 16#9AB4;
   // UNICODE_TO_GBK[16720] := 16#6BDB;
   // UNICODE_TO_GBK[16721] := 16#C3AB;
   // UNICODE_TO_GBK[16722] := 16#6BDC;
   // UNICODE_TO_GBK[16723] := 16#9AB5;
   // UNICODE_TO_GBK[16724] := 16#6BDD;
   // UNICODE_TO_GBK[16725] := 16#9AB6;
   // UNICODE_TO_GBK[16726] := 16#6BDE;
   // UNICODE_TO_GBK[16727] := 16#9AB7;
   // UNICODE_TO_GBK[16728] := 16#6BDF;
   // UNICODE_TO_GBK[16729] := 16#9AB8;
   // UNICODE_TO_GBK[16730] := 16#6BE0;
   // UNICODE_TO_GBK[16731] := 16#9AB9;
   // UNICODE_TO_GBK[16732] := 16#6BE1;
   // UNICODE_TO_GBK[16733] := 16#D5B1;
   // UNICODE_TO_GBK[16734] := 16#6BE2;
   // UNICODE_TO_GBK[16735] := 16#9ABA;
   // UNICODE_TO_GBK[16736] := 16#6BE3;
   // UNICODE_TO_GBK[16737] := 16#9ABB;
   // UNICODE_TO_GBK[16738] := 16#6BE4;
   // UNICODE_TO_GBK[16739] := 16#9ABC;
   // UNICODE_TO_GBK[16740] := 16#6BE5;
   // UNICODE_TO_GBK[16741] := 16#9ABD;
   // UNICODE_TO_GBK[16742] := 16#6BE6;
   // UNICODE_TO_GBK[16743] := 16#9ABE;
   // UNICODE_TO_GBK[16744] := 16#6BE7;
   // UNICODE_TO_GBK[16745] := 16#9ABF;
   // UNICODE_TO_GBK[16746] := 16#6BE8;
   // UNICODE_TO_GBK[16747] := 16#9AC0;
   // UNICODE_TO_GBK[16748] := 16#6BE9;
   // UNICODE_TO_GBK[16749] := 16#9AC1;
   // UNICODE_TO_GBK[16750] := 16#6BEA;
   // UNICODE_TO_GBK[16751] := 16#EBA4;
   // UNICODE_TO_GBK[16752] := 16#6BEB;
   // UNICODE_TO_GBK[16753] := 16#BAC1;
   // UNICODE_TO_GBK[16754] := 16#6BEC;
   // UNICODE_TO_GBK[16755] := 16#9AC2;
   // UNICODE_TO_GBK[16756] := 16#6BED;
   // UNICODE_TO_GBK[16757] := 16#9AC3;
   // UNICODE_TO_GBK[16758] := 16#6BEE;
   // UNICODE_TO_GBK[16759] := 16#9AC4;
   // UNICODE_TO_GBK[16760] := 16#6BEF;
   // UNICODE_TO_GBK[16761] := 16#CCBA;
   // UNICODE_TO_GBK[16762] := 16#6BF0;
   // UNICODE_TO_GBK[16763] := 16#9AC5;
   // UNICODE_TO_GBK[16764] := 16#6BF1;
   // UNICODE_TO_GBK[16765] := 16#9AC6;
   // UNICODE_TO_GBK[16766] := 16#6BF2;
   // UNICODE_TO_GBK[16767] := 16#9AC7;
   // UNICODE_TO_GBK[16768] := 16#6BF3;
   // UNICODE_TO_GBK[16769] := 16#EBA5;
   // UNICODE_TO_GBK[16770] := 16#6BF4;
   // UNICODE_TO_GBK[16771] := 16#9AC8;
   // UNICODE_TO_GBK[16772] := 16#6BF5;
   // UNICODE_TO_GBK[16773] := 16#EBA7;
   // UNICODE_TO_GBK[16774] := 16#6BF6;
   // UNICODE_TO_GBK[16775] := 16#9AC9;
   // UNICODE_TO_GBK[16776] := 16#6BF7;
   // UNICODE_TO_GBK[16777] := 16#9ACA;
   // UNICODE_TO_GBK[16778] := 16#6BF8;
   // UNICODE_TO_GBK[16779] := 16#9ACB;
   // UNICODE_TO_GBK[16780] := 16#6BF9;
   // UNICODE_TO_GBK[16781] := 16#EBA8;
   // UNICODE_TO_GBK[16782] := 16#6BFA;
   // UNICODE_TO_GBK[16783] := 16#9ACC;
   // UNICODE_TO_GBK[16784] := 16#6BFB;
   // UNICODE_TO_GBK[16785] := 16#9ACD;
   // UNICODE_TO_GBK[16786] := 16#6BFC;
   // UNICODE_TO_GBK[16787] := 16#9ACE;
   // UNICODE_TO_GBK[16788] := 16#6BFD;
   // UNICODE_TO_GBK[16789] := 16#EBA6;
   // UNICODE_TO_GBK[16790] := 16#6BFE;
   // UNICODE_TO_GBK[16791] := 16#9ACF;
   // UNICODE_TO_GBK[16792] := 16#6BFF;
   // UNICODE_TO_GBK[16793] := 16#9AD0;
   // UNICODE_TO_GBK[16794] := 16#6C00;
   // UNICODE_TO_GBK[16795] := 16#9AD1;
   // UNICODE_TO_GBK[16796] := 16#6C01;
   // UNICODE_TO_GBK[16797] := 16#9AD2;
   // UNICODE_TO_GBK[16798] := 16#6C02;
   // UNICODE_TO_GBK[16799] := 16#9AD3;
   // UNICODE_TO_GBK[16800] := 16#6C03;
   // UNICODE_TO_GBK[16801] := 16#9AD4;
   // UNICODE_TO_GBK[16802] := 16#6C04;
   // UNICODE_TO_GBK[16803] := 16#9AD5;
   // UNICODE_TO_GBK[16804] := 16#6C05;
   // UNICODE_TO_GBK[16805] := 16#EBA9;
   // UNICODE_TO_GBK[16806] := 16#6C06;
   // UNICODE_TO_GBK[16807] := 16#EBAB;
   // UNICODE_TO_GBK[16808] := 16#6C07;
   // UNICODE_TO_GBK[16809] := 16#EBAA;
   // UNICODE_TO_GBK[16810] := 16#6C08;
   // UNICODE_TO_GBK[16811] := 16#9AD6;
   // UNICODE_TO_GBK[16812] := 16#6C09;
   // UNICODE_TO_GBK[16813] := 16#9AD7;
   // UNICODE_TO_GBK[16814] := 16#6C0A;
   // UNICODE_TO_GBK[16815] := 16#9AD8;
   // UNICODE_TO_GBK[16816] := 16#6C0B;
   // UNICODE_TO_GBK[16817] := 16#9AD9;
   // UNICODE_TO_GBK[16818] := 16#6C0C;
   // UNICODE_TO_GBK[16819] := 16#9ADA;
   // UNICODE_TO_GBK[16820] := 16#6C0D;
   // UNICODE_TO_GBK[16821] := 16#EBAC;
   // UNICODE_TO_GBK[16822] := 16#6C0E;
   // UNICODE_TO_GBK[16823] := 16#9ADB;
   // UNICODE_TO_GBK[16824] := 16#6C0F;
   // UNICODE_TO_GBK[16825] := 16#CACF;
   // UNICODE_TO_GBK[16826] := 16#6C10;
   // UNICODE_TO_GBK[16827] := 16#D8B5;
   // UNICODE_TO_GBK[16828] := 16#6C11;
   // UNICODE_TO_GBK[16829] := 16#C3F1;
   // UNICODE_TO_GBK[16830] := 16#6C12;
   // UNICODE_TO_GBK[16831] := 16#9ADC;
   // UNICODE_TO_GBK[16832] := 16#6C13;
   // UNICODE_TO_GBK[16833] := 16#C3A5;
   // UNICODE_TO_GBK[16834] := 16#6C14;
   // UNICODE_TO_GBK[16835] := 16#C6F8;
   // UNICODE_TO_GBK[16836] := 16#6C15;
   // UNICODE_TO_GBK[16837] := 16#EBAD;
   // UNICODE_TO_GBK[16838] := 16#6C16;
   // UNICODE_TO_GBK[16839] := 16#C4CA;
   // UNICODE_TO_GBK[16840] := 16#6C17;
   // UNICODE_TO_GBK[16841] := 16#9ADD;
   // UNICODE_TO_GBK[16842] := 16#6C18;
   // UNICODE_TO_GBK[16843] := 16#EBAE;
   // UNICODE_TO_GBK[16844] := 16#6C19;
   // UNICODE_TO_GBK[16845] := 16#EBAF;
   // UNICODE_TO_GBK[16846] := 16#6C1A;
   // UNICODE_TO_GBK[16847] := 16#EBB0;
   // UNICODE_TO_GBK[16848] := 16#6C1B;
   // UNICODE_TO_GBK[16849] := 16#B7D5;
   // UNICODE_TO_GBK[16850] := 16#6C1C;
   // UNICODE_TO_GBK[16851] := 16#9ADE;
   // UNICODE_TO_GBK[16852] := 16#6C1D;
   // UNICODE_TO_GBK[16853] := 16#9ADF;
   // UNICODE_TO_GBK[16854] := 16#6C1E;
   // UNICODE_TO_GBK[16855] := 16#9AE0;
   // UNICODE_TO_GBK[16856] := 16#6C1F;
   // UNICODE_TO_GBK[16857] := 16#B7FA;
   // UNICODE_TO_GBK[16858] := 16#6C20;
   // UNICODE_TO_GBK[16859] := 16#9AE1;
   // UNICODE_TO_GBK[16860] := 16#6C21;
   // UNICODE_TO_GBK[16861] := 16#EBB1;
   // UNICODE_TO_GBK[16862] := 16#6C22;
   // UNICODE_TO_GBK[16863] := 16#C7E2;
   // UNICODE_TO_GBK[16864] := 16#6C23;
   // UNICODE_TO_GBK[16865] := 16#9AE2;
   // UNICODE_TO_GBK[16866] := 16#6C24;
   // UNICODE_TO_GBK[16867] := 16#EBB3;
   // UNICODE_TO_GBK[16868] := 16#6C25;
   // UNICODE_TO_GBK[16869] := 16#9AE3;
   // UNICODE_TO_GBK[16870] := 16#6C26;
   // UNICODE_TO_GBK[16871] := 16#BAA4;
   // UNICODE_TO_GBK[16872] := 16#6C27;
   // UNICODE_TO_GBK[16873] := 16#D1F5;
   // UNICODE_TO_GBK[16874] := 16#6C28;
   // UNICODE_TO_GBK[16875] := 16#B0B1;
   // UNICODE_TO_GBK[16876] := 16#6C29;
   // UNICODE_TO_GBK[16877] := 16#EBB2;
   // UNICODE_TO_GBK[16878] := 16#6C2A;
   // UNICODE_TO_GBK[16879] := 16#EBB4;
   // UNICODE_TO_GBK[16880] := 16#6C2B;
   // UNICODE_TO_GBK[16881] := 16#9AE4;
   // UNICODE_TO_GBK[16882] := 16#6C2C;
   // UNICODE_TO_GBK[16883] := 16#9AE5;
   // UNICODE_TO_GBK[16884] := 16#6C2D;
   // UNICODE_TO_GBK[16885] := 16#9AE6;
   // UNICODE_TO_GBK[16886] := 16#6C2E;
   // UNICODE_TO_GBK[16887] := 16#B5AA;
   // UNICODE_TO_GBK[16888] := 16#6C2F;
   // UNICODE_TO_GBK[16889] := 16#C2C8;
   // UNICODE_TO_GBK[16890] := 16#6C30;
   // UNICODE_TO_GBK[16891] := 16#C7E8;
   // UNICODE_TO_GBK[16892] := 16#6C31;
   // UNICODE_TO_GBK[16893] := 16#9AE7;
   // UNICODE_TO_GBK[16894] := 16#6C32;
   // UNICODE_TO_GBK[16895] := 16#EBB5;
   // UNICODE_TO_GBK[16896] := 16#6C33;
   // UNICODE_TO_GBK[16897] := 16#9AE8;
   // UNICODE_TO_GBK[16898] := 16#6C34;
   // UNICODE_TO_GBK[16899] := 16#CBAE;
   // UNICODE_TO_GBK[16900] := 16#6C35;
   // UNICODE_TO_GBK[16901] := 16#E3DF;
   // UNICODE_TO_GBK[16902] := 16#6C36;
   // UNICODE_TO_GBK[16903] := 16#9AE9;
   // UNICODE_TO_GBK[16904] := 16#6C37;
   // UNICODE_TO_GBK[16905] := 16#9AEA;
   // UNICODE_TO_GBK[16906] := 16#6C38;
   // UNICODE_TO_GBK[16907] := 16#D3C0;
   // UNICODE_TO_GBK[16908] := 16#6C39;
   // UNICODE_TO_GBK[16909] := 16#9AEB;
   // UNICODE_TO_GBK[16910] := 16#6C3A;
   // UNICODE_TO_GBK[16911] := 16#9AEC;
   // UNICODE_TO_GBK[16912] := 16#6C3B;
   // UNICODE_TO_GBK[16913] := 16#9AED;
   // UNICODE_TO_GBK[16914] := 16#6C3C;
   // UNICODE_TO_GBK[16915] := 16#9AEE;
   // UNICODE_TO_GBK[16916] := 16#6C3D;
   // UNICODE_TO_GBK[16917] := 16#D9DB;
   // UNICODE_TO_GBK[16918] := 16#6C3E;
   // UNICODE_TO_GBK[16919] := 16#9AEF;
   // UNICODE_TO_GBK[16920] := 16#6C3F;
   // UNICODE_TO_GBK[16921] := 16#9AF0;
   // UNICODE_TO_GBK[16922] := 16#6C40;
   // UNICODE_TO_GBK[16923] := 16#CDA1;
   // UNICODE_TO_GBK[16924] := 16#6C41;
   // UNICODE_TO_GBK[16925] := 16#D6AD;
   // UNICODE_TO_GBK[16926] := 16#6C42;
   // UNICODE_TO_GBK[16927] := 16#C7F3;
   // UNICODE_TO_GBK[16928] := 16#6C43;
   // UNICODE_TO_GBK[16929] := 16#9AF1;
   // UNICODE_TO_GBK[16930] := 16#6C44;
   // UNICODE_TO_GBK[16931] := 16#9AF2;
   // UNICODE_TO_GBK[16932] := 16#6C45;
   // UNICODE_TO_GBK[16933] := 16#9AF3;
   // UNICODE_TO_GBK[16934] := 16#6C46;
   // UNICODE_TO_GBK[16935] := 16#D9E0;
   // UNICODE_TO_GBK[16936] := 16#6C47;
   // UNICODE_TO_GBK[16937] := 16#BBE3;
   // UNICODE_TO_GBK[16938] := 16#6C48;
   // UNICODE_TO_GBK[16939] := 16#9AF4;
   // UNICODE_TO_GBK[16940] := 16#6C49;
   // UNICODE_TO_GBK[16941] := 16#BABA;
   // UNICODE_TO_GBK[16942] := 16#6C4A;
   // UNICODE_TO_GBK[16943] := 16#E3E2;
   // UNICODE_TO_GBK[16944] := 16#6C4B;
   // UNICODE_TO_GBK[16945] := 16#9AF5;
   // UNICODE_TO_GBK[16946] := 16#6C4C;
   // UNICODE_TO_GBK[16947] := 16#9AF6;
   // UNICODE_TO_GBK[16948] := 16#6C4D;
   // UNICODE_TO_GBK[16949] := 16#9AF7;
   // UNICODE_TO_GBK[16950] := 16#6C4E;
   // UNICODE_TO_GBK[16951] := 16#9AF8;
   // UNICODE_TO_GBK[16952] := 16#6C4F;
   // UNICODE_TO_GBK[16953] := 16#9AF9;
   // UNICODE_TO_GBK[16954] := 16#6C50;
   // UNICODE_TO_GBK[16955] := 16#CFAB;
   // UNICODE_TO_GBK[16956] := 16#6C51;
   // UNICODE_TO_GBK[16957] := 16#9AFA;
   // UNICODE_TO_GBK[16958] := 16#6C52;
   // UNICODE_TO_GBK[16959] := 16#9AFB;
   // UNICODE_TO_GBK[16960] := 16#6C53;
   // UNICODE_TO_GBK[16961] := 16#9AFC;
   // UNICODE_TO_GBK[16962] := 16#6C54;
   // UNICODE_TO_GBK[16963] := 16#E3E0;
   // UNICODE_TO_GBK[16964] := 16#6C55;
   // UNICODE_TO_GBK[16965] := 16#C9C7;
   // UNICODE_TO_GBK[16966] := 16#6C56;
   // UNICODE_TO_GBK[16967] := 16#9AFD;
   // UNICODE_TO_GBK[16968] := 16#6C57;
   // UNICODE_TO_GBK[16969] := 16#BAB9;
   // UNICODE_TO_GBK[16970] := 16#6C58;
   // UNICODE_TO_GBK[16971] := 16#9AFE;
   // UNICODE_TO_GBK[16972] := 16#6C59;
   // UNICODE_TO_GBK[16973] := 16#9B40;
   // UNICODE_TO_GBK[16974] := 16#6C5A;
   // UNICODE_TO_GBK[16975] := 16#9B41;
   // UNICODE_TO_GBK[16976] := 16#6C5B;
   // UNICODE_TO_GBK[16977] := 16#D1B4;
   // UNICODE_TO_GBK[16978] := 16#6C5C;
   // UNICODE_TO_GBK[16979] := 16#E3E1;
   // UNICODE_TO_GBK[16980] := 16#6C5D;
   // UNICODE_TO_GBK[16981] := 16#C8EA;
   // UNICODE_TO_GBK[16982] := 16#6C5E;
   // UNICODE_TO_GBK[16983] := 16#B9AF;
   // UNICODE_TO_GBK[16984] := 16#6C5F;
   // UNICODE_TO_GBK[16985] := 16#BDAD;
   // UNICODE_TO_GBK[16986] := 16#6C60;
   // UNICODE_TO_GBK[16987] := 16#B3D8;
   // UNICODE_TO_GBK[16988] := 16#6C61;
   // UNICODE_TO_GBK[16989] := 16#CEDB;
   // UNICODE_TO_GBK[16990] := 16#6C62;
   // UNICODE_TO_GBK[16991] := 16#9B42;
   // UNICODE_TO_GBK[16992] := 16#6C63;
   // UNICODE_TO_GBK[16993] := 16#9B43;
   // UNICODE_TO_GBK[16994] := 16#6C64;
   // UNICODE_TO_GBK[16995] := 16#CCC0;
   // UNICODE_TO_GBK[16996] := 16#6C65;
   // UNICODE_TO_GBK[16997] := 16#9B44;
   // UNICODE_TO_GBK[16998] := 16#6C66;
   // UNICODE_TO_GBK[16999] := 16#9B45;
   // UNICODE_TO_GBK[17000] := 16#6C67;
   // UNICODE_TO_GBK[17001] := 16#9B46;
   // UNICODE_TO_GBK[17002] := 16#6C68;
   // UNICODE_TO_GBK[17003] := 16#E3E8;
   // UNICODE_TO_GBK[17004] := 16#6C69;
   // UNICODE_TO_GBK[17005] := 16#E3E9;
   // UNICODE_TO_GBK[17006] := 16#6C6A;
   // UNICODE_TO_GBK[17007] := 16#CDF4;
   // UNICODE_TO_GBK[17008] := 16#6C6B;
   // UNICODE_TO_GBK[17009] := 16#9B47;
   // UNICODE_TO_GBK[17010] := 16#6C6C;
   // UNICODE_TO_GBK[17011] := 16#9B48;
   // UNICODE_TO_GBK[17012] := 16#6C6D;
   // UNICODE_TO_GBK[17013] := 16#9B49;
   // UNICODE_TO_GBK[17014] := 16#6C6E;
   // UNICODE_TO_GBK[17015] := 16#9B4A;
   // UNICODE_TO_GBK[17016] := 16#6C6F;
   // UNICODE_TO_GBK[17017] := 16#9B4B;
   // UNICODE_TO_GBK[17018] := 16#6C70;
   // UNICODE_TO_GBK[17019] := 16#CCAD;
   // UNICODE_TO_GBK[17020] := 16#6C71;
   // UNICODE_TO_GBK[17021] := 16#9B4C;
   // UNICODE_TO_GBK[17022] := 16#6C72;
   // UNICODE_TO_GBK[17023] := 16#BCB3;
   // UNICODE_TO_GBK[17024] := 16#6C73;
   // UNICODE_TO_GBK[17025] := 16#9B4D;
   // UNICODE_TO_GBK[17026] := 16#6C74;
   // UNICODE_TO_GBK[17027] := 16#E3EA;
   // UNICODE_TO_GBK[17028] := 16#6C75;
   // UNICODE_TO_GBK[17029] := 16#9B4E;
   // UNICODE_TO_GBK[17030] := 16#6C76;
   // UNICODE_TO_GBK[17031] := 16#E3EB;
   // UNICODE_TO_GBK[17032] := 16#6C77;
   // UNICODE_TO_GBK[17033] := 16#9B4F;
   // UNICODE_TO_GBK[17034] := 16#6C78;
   // UNICODE_TO_GBK[17035] := 16#9B50;
   // UNICODE_TO_GBK[17036] := 16#6C79;
   // UNICODE_TO_GBK[17037] := 16#D0DA;
   // UNICODE_TO_GBK[17038] := 16#6C7A;
   // UNICODE_TO_GBK[17039] := 16#9B51;
   // UNICODE_TO_GBK[17040] := 16#6C7B;
   // UNICODE_TO_GBK[17041] := 16#9B52;
   // UNICODE_TO_GBK[17042] := 16#6C7C;
   // UNICODE_TO_GBK[17043] := 16#9B53;
   // UNICODE_TO_GBK[17044] := 16#6C7D;
   // UNICODE_TO_GBK[17045] := 16#C6FB;
   // UNICODE_TO_GBK[17046] := 16#6C7E;
   // UNICODE_TO_GBK[17047] := 16#B7DA;
   // UNICODE_TO_GBK[17048] := 16#6C7F;
   // UNICODE_TO_GBK[17049] := 16#9B54;
   // UNICODE_TO_GBK[17050] := 16#6C80;
   // UNICODE_TO_GBK[17051] := 16#9B55;
   // UNICODE_TO_GBK[17052] := 16#6C81;
   // UNICODE_TO_GBK[17053] := 16#C7DF;
   // UNICODE_TO_GBK[17054] := 16#6C82;
   // UNICODE_TO_GBK[17055] := 16#D2CA;
   // UNICODE_TO_GBK[17056] := 16#6C83;
   // UNICODE_TO_GBK[17057] := 16#CED6;
   // UNICODE_TO_GBK[17058] := 16#6C84;
   // UNICODE_TO_GBK[17059] := 16#9B56;
   // UNICODE_TO_GBK[17060] := 16#6C85;
   // UNICODE_TO_GBK[17061] := 16#E3E4;
   // UNICODE_TO_GBK[17062] := 16#6C86;
   // UNICODE_TO_GBK[17063] := 16#E3EC;
   // UNICODE_TO_GBK[17064] := 16#6C87;
   // UNICODE_TO_GBK[17065] := 16#9B57;
   // UNICODE_TO_GBK[17066] := 16#6C88;
   // UNICODE_TO_GBK[17067] := 16#C9F2;
   // UNICODE_TO_GBK[17068] := 16#6C89;
   // UNICODE_TO_GBK[17069] := 16#B3C1;
   // UNICODE_TO_GBK[17070] := 16#6C8A;
   // UNICODE_TO_GBK[17071] := 16#9B58;
   // UNICODE_TO_GBK[17072] := 16#6C8B;
   // UNICODE_TO_GBK[17073] := 16#9B59;
   // UNICODE_TO_GBK[17074] := 16#6C8C;
   // UNICODE_TO_GBK[17075] := 16#E3E7;
   // UNICODE_TO_GBK[17076] := 16#6C8D;
   // UNICODE_TO_GBK[17077] := 16#9B5A;
   // UNICODE_TO_GBK[17078] := 16#6C8E;
   // UNICODE_TO_GBK[17079] := 16#9B5B;
   // UNICODE_TO_GBK[17080] := 16#6C8F;
   // UNICODE_TO_GBK[17081] := 16#C6E3;
   // UNICODE_TO_GBK[17082] := 16#6C90;
   // UNICODE_TO_GBK[17083] := 16#E3E5;
   // UNICODE_TO_GBK[17084] := 16#6C91;
   // UNICODE_TO_GBK[17085] := 16#9B5C;
   // UNICODE_TO_GBK[17086] := 16#6C92;
   // UNICODE_TO_GBK[17087] := 16#9B5D;
   // UNICODE_TO_GBK[17088] := 16#6C93;
   // UNICODE_TO_GBK[17089] := 16#EDB3;
   // UNICODE_TO_GBK[17090] := 16#6C94;
   // UNICODE_TO_GBK[17091] := 16#E3E6;
   // UNICODE_TO_GBK[17092] := 16#6C95;
   // UNICODE_TO_GBK[17093] := 16#9B5E;
   // UNICODE_TO_GBK[17094] := 16#6C96;
   // UNICODE_TO_GBK[17095] := 16#9B5F;
   // UNICODE_TO_GBK[17096] := 16#6C97;
   // UNICODE_TO_GBK[17097] := 16#9B60;
   // UNICODE_TO_GBK[17098] := 16#6C98;
   // UNICODE_TO_GBK[17099] := 16#9B61;
   // UNICODE_TO_GBK[17100] := 16#6C99;
   // UNICODE_TO_GBK[17101] := 16#C9B3;
   // UNICODE_TO_GBK[17102] := 16#6C9A;
   // UNICODE_TO_GBK[17103] := 16#9B62;
   // UNICODE_TO_GBK[17104] := 16#6C9B;
   // UNICODE_TO_GBK[17105] := 16#C5E6;
   // UNICODE_TO_GBK[17106] := 16#6C9C;
   // UNICODE_TO_GBK[17107] := 16#9B63;
   // UNICODE_TO_GBK[17108] := 16#6C9D;
   // UNICODE_TO_GBK[17109] := 16#9B64;
   // UNICODE_TO_GBK[17110] := 16#6C9E;
   // UNICODE_TO_GBK[17111] := 16#9B65;
   // UNICODE_TO_GBK[17112] := 16#6C9F;
   // UNICODE_TO_GBK[17113] := 16#B9B5;
   // UNICODE_TO_GBK[17114] := 16#6CA0;
   // UNICODE_TO_GBK[17115] := 16#9B66;
   // UNICODE_TO_GBK[17116] := 16#6CA1;
   // UNICODE_TO_GBK[17117] := 16#C3BB;
   // UNICODE_TO_GBK[17118] := 16#6CA2;
   // UNICODE_TO_GBK[17119] := 16#9B67;
   // UNICODE_TO_GBK[17120] := 16#6CA3;
   // UNICODE_TO_GBK[17121] := 16#E3E3;
   // UNICODE_TO_GBK[17122] := 16#6CA4;
   // UNICODE_TO_GBK[17123] := 16#C5BD;
   // UNICODE_TO_GBK[17124] := 16#6CA5;
   // UNICODE_TO_GBK[17125] := 16#C1A4;
   // UNICODE_TO_GBK[17126] := 16#6CA6;
   // UNICODE_TO_GBK[17127] := 16#C2D9;
   // UNICODE_TO_GBK[17128] := 16#6CA7;
   // UNICODE_TO_GBK[17129] := 16#B2D7;
   // UNICODE_TO_GBK[17130] := 16#6CA8;
   // UNICODE_TO_GBK[17131] := 16#9B68;
   // UNICODE_TO_GBK[17132] := 16#6CA9;
   // UNICODE_TO_GBK[17133] := 16#E3ED;
   // UNICODE_TO_GBK[17134] := 16#6CAA;
   // UNICODE_TO_GBK[17135] := 16#BBA6;
   // UNICODE_TO_GBK[17136] := 16#6CAB;
   // UNICODE_TO_GBK[17137] := 16#C4AD;
   // UNICODE_TO_GBK[17138] := 16#6CAC;
   // UNICODE_TO_GBK[17139] := 16#9B69;
   // UNICODE_TO_GBK[17140] := 16#6CAD;
   // UNICODE_TO_GBK[17141] := 16#E3F0;
   // UNICODE_TO_GBK[17142] := 16#6CAE;
   // UNICODE_TO_GBK[17143] := 16#BEDA;
   // UNICODE_TO_GBK[17144] := 16#6CAF;
   // UNICODE_TO_GBK[17145] := 16#9B6A;
   // UNICODE_TO_GBK[17146] := 16#6CB0;
   // UNICODE_TO_GBK[17147] := 16#9B6B;
   // UNICODE_TO_GBK[17148] := 16#6CB1;
   // UNICODE_TO_GBK[17149] := 16#E3FB;
   // UNICODE_TO_GBK[17150] := 16#6CB2;
   // UNICODE_TO_GBK[17151] := 16#E3F5;
   // UNICODE_TO_GBK[17152] := 16#6CB3;
   // UNICODE_TO_GBK[17153] := 16#BAD3;
   // UNICODE_TO_GBK[17154] := 16#6CB4;
   // UNICODE_TO_GBK[17155] := 16#9B6C;
   // UNICODE_TO_GBK[17156] := 16#6CB5;
   // UNICODE_TO_GBK[17157] := 16#9B6D;
   // UNICODE_TO_GBK[17158] := 16#6CB6;
   // UNICODE_TO_GBK[17159] := 16#9B6E;
   // UNICODE_TO_GBK[17160] := 16#6CB7;
   // UNICODE_TO_GBK[17161] := 16#9B6F;
   // UNICODE_TO_GBK[17162] := 16#6CB8;
   // UNICODE_TO_GBK[17163] := 16#B7D0;
   // UNICODE_TO_GBK[17164] := 16#6CB9;
   // UNICODE_TO_GBK[17165] := 16#D3CD;
   // UNICODE_TO_GBK[17166] := 16#6CBA;
   // UNICODE_TO_GBK[17167] := 16#9B70;
   // UNICODE_TO_GBK[17168] := 16#6CBB;
   // UNICODE_TO_GBK[17169] := 16#D6CE;
   // UNICODE_TO_GBK[17170] := 16#6CBC;
   // UNICODE_TO_GBK[17171] := 16#D5D3;
   // UNICODE_TO_GBK[17172] := 16#6CBD;
   // UNICODE_TO_GBK[17173] := 16#B9C1;
   // UNICODE_TO_GBK[17174] := 16#6CBE;
   // UNICODE_TO_GBK[17175] := 16#D5B4;
   // UNICODE_TO_GBK[17176] := 16#6CBF;
   // UNICODE_TO_GBK[17177] := 16#D1D8;
   // UNICODE_TO_GBK[17178] := 16#6CC0;
   // UNICODE_TO_GBK[17179] := 16#9B71;
   // UNICODE_TO_GBK[17180] := 16#6CC1;
   // UNICODE_TO_GBK[17181] := 16#9B72;
   // UNICODE_TO_GBK[17182] := 16#6CC2;
   // UNICODE_TO_GBK[17183] := 16#9B73;
   // UNICODE_TO_GBK[17184] := 16#6CC3;
   // UNICODE_TO_GBK[17185] := 16#9B74;
   // UNICODE_TO_GBK[17186] := 16#6CC4;
   // UNICODE_TO_GBK[17187] := 16#D0B9;
   // UNICODE_TO_GBK[17188] := 16#6CC5;
   // UNICODE_TO_GBK[17189] := 16#C7F6;
   // UNICODE_TO_GBK[17190] := 16#6CC6;
   // UNICODE_TO_GBK[17191] := 16#9B75;
   // UNICODE_TO_GBK[17192] := 16#6CC7;
   // UNICODE_TO_GBK[17193] := 16#9B76;
   // UNICODE_TO_GBK[17194] := 16#6CC8;
   // UNICODE_TO_GBK[17195] := 16#9B77;
   // UNICODE_TO_GBK[17196] := 16#6CC9;
   // UNICODE_TO_GBK[17197] := 16#C8AA;
   // UNICODE_TO_GBK[17198] := 16#6CCA;
   // UNICODE_TO_GBK[17199] := 16#B2B4;
   // UNICODE_TO_GBK[17200] := 16#6CCB;
   // UNICODE_TO_GBK[17201] := 16#9B78;
   // UNICODE_TO_GBK[17202] := 16#6CCC;
   // UNICODE_TO_GBK[17203] := 16#C3DA;
   // UNICODE_TO_GBK[17204] := 16#6CCD;
   // UNICODE_TO_GBK[17205] := 16#9B79;
   // UNICODE_TO_GBK[17206] := 16#6CCE;
   // UNICODE_TO_GBK[17207] := 16#9B7A;
   // UNICODE_TO_GBK[17208] := 16#6CCF;
   // UNICODE_TO_GBK[17209] := 16#9B7B;
   // UNICODE_TO_GBK[17210] := 16#6CD0;
   // UNICODE_TO_GBK[17211] := 16#E3EE;
   // UNICODE_TO_GBK[17212] := 16#6CD1;
   // UNICODE_TO_GBK[17213] := 16#9B7C;
   // UNICODE_TO_GBK[17214] := 16#6CD2;
   // UNICODE_TO_GBK[17215] := 16#9B7D;
   // UNICODE_TO_GBK[17216] := 16#6CD3;
   // UNICODE_TO_GBK[17217] := 16#E3FC;
   // UNICODE_TO_GBK[17218] := 16#6CD4;
   // UNICODE_TO_GBK[17219] := 16#E3EF;
   // UNICODE_TO_GBK[17220] := 16#6CD5;
   // UNICODE_TO_GBK[17221] := 16#B7A8;
   // UNICODE_TO_GBK[17222] := 16#6CD6;
   // UNICODE_TO_GBK[17223] := 16#E3F7;
   // UNICODE_TO_GBK[17224] := 16#6CD7;
   // UNICODE_TO_GBK[17225] := 16#E3F4;
   // UNICODE_TO_GBK[17226] := 16#6CD8;
   // UNICODE_TO_GBK[17227] := 16#9B7E;
   // UNICODE_TO_GBK[17228] := 16#6CD9;
   // UNICODE_TO_GBK[17229] := 16#9B80;
   // UNICODE_TO_GBK[17230] := 16#6CDA;
   // UNICODE_TO_GBK[17231] := 16#9B81;
   // UNICODE_TO_GBK[17232] := 16#6CDB;
   // UNICODE_TO_GBK[17233] := 16#B7BA;
   // UNICODE_TO_GBK[17234] := 16#6CDC;
   // UNICODE_TO_GBK[17235] := 16#9B82;
   // UNICODE_TO_GBK[17236] := 16#6CDD;
   // UNICODE_TO_GBK[17237] := 16#9B83;
   // UNICODE_TO_GBK[17238] := 16#6CDE;
   // UNICODE_TO_GBK[17239] := 16#C5A2;
   // UNICODE_TO_GBK[17240] := 16#6CDF;
   // UNICODE_TO_GBK[17241] := 16#9B84;
   // UNICODE_TO_GBK[17242] := 16#6CE0;
   // UNICODE_TO_GBK[17243] := 16#E3F6;
   // UNICODE_TO_GBK[17244] := 16#6CE1;
   // UNICODE_TO_GBK[17245] := 16#C5DD;
   // UNICODE_TO_GBK[17246] := 16#6CE2;
   // UNICODE_TO_GBK[17247] := 16#B2A8;
   // UNICODE_TO_GBK[17248] := 16#6CE3;
   // UNICODE_TO_GBK[17249] := 16#C6FC;
   // UNICODE_TO_GBK[17250] := 16#6CE4;
   // UNICODE_TO_GBK[17251] := 16#9B85;
   // UNICODE_TO_GBK[17252] := 16#6CE5;
   // UNICODE_TO_GBK[17253] := 16#C4E0;
   // UNICODE_TO_GBK[17254] := 16#6CE6;
   // UNICODE_TO_GBK[17255] := 16#9B86;
   // UNICODE_TO_GBK[17256] := 16#6CE7;
   // UNICODE_TO_GBK[17257] := 16#9B87;
   // UNICODE_TO_GBK[17258] := 16#6CE8;
   // UNICODE_TO_GBK[17259] := 16#D7A2;
   // UNICODE_TO_GBK[17260] := 16#6CE9;
   // UNICODE_TO_GBK[17261] := 16#9B88;
   // UNICODE_TO_GBK[17262] := 16#6CEA;
   // UNICODE_TO_GBK[17263] := 16#C0E1;
   // UNICODE_TO_GBK[17264] := 16#6CEB;
   // UNICODE_TO_GBK[17265] := 16#E3F9;
   // UNICODE_TO_GBK[17266] := 16#6CEC;
   // UNICODE_TO_GBK[17267] := 16#9B89;
   // UNICODE_TO_GBK[17268] := 16#6CED;
   // UNICODE_TO_GBK[17269] := 16#9B8A;
   // UNICODE_TO_GBK[17270] := 16#6CEE;
   // UNICODE_TO_GBK[17271] := 16#E3FA;
   // UNICODE_TO_GBK[17272] := 16#6CEF;
   // UNICODE_TO_GBK[17273] := 16#E3FD;
   // UNICODE_TO_GBK[17274] := 16#6CF0;
   // UNICODE_TO_GBK[17275] := 16#CCA9;
   // UNICODE_TO_GBK[17276] := 16#6CF1;
   // UNICODE_TO_GBK[17277] := 16#E3F3;
   // UNICODE_TO_GBK[17278] := 16#6CF2;
   // UNICODE_TO_GBK[17279] := 16#9B8B;
   // UNICODE_TO_GBK[17280] := 16#6CF3;
   // UNICODE_TO_GBK[17281] := 16#D3BE;
   // UNICODE_TO_GBK[17282] := 16#6CF4;
   // UNICODE_TO_GBK[17283] := 16#9B8C;
   // UNICODE_TO_GBK[17284] := 16#6CF5;
   // UNICODE_TO_GBK[17285] := 16#B1C3;
   // UNICODE_TO_GBK[17286] := 16#6CF6;
   // UNICODE_TO_GBK[17287] := 16#EDB4;
   // UNICODE_TO_GBK[17288] := 16#6CF7;
   // UNICODE_TO_GBK[17289] := 16#E3F1;
   // UNICODE_TO_GBK[17290] := 16#6CF8;
   // UNICODE_TO_GBK[17291] := 16#E3F2;
   // UNICODE_TO_GBK[17292] := 16#6CF9;
   // UNICODE_TO_GBK[17293] := 16#9B8D;
   // UNICODE_TO_GBK[17294] := 16#6CFA;
   // UNICODE_TO_GBK[17295] := 16#E3F8;
   // UNICODE_TO_GBK[17296] := 16#6CFB;
   // UNICODE_TO_GBK[17297] := 16#D0BA;
   // UNICODE_TO_GBK[17298] := 16#6CFC;
   // UNICODE_TO_GBK[17299] := 16#C6C3;
   // UNICODE_TO_GBK[17300] := 16#6CFD;
   // UNICODE_TO_GBK[17301] := 16#D4F3;
   // UNICODE_TO_GBK[17302] := 16#6CFE;
   // UNICODE_TO_GBK[17303] := 16#E3FE;
   // UNICODE_TO_GBK[17304] := 16#6CFF;
   // UNICODE_TO_GBK[17305] := 16#9B8E;
   // UNICODE_TO_GBK[17306] := 16#6D00;
   // UNICODE_TO_GBK[17307] := 16#9B8F;
   // UNICODE_TO_GBK[17308] := 16#6D01;
   // UNICODE_TO_GBK[17309] := 16#BDE0;
   // UNICODE_TO_GBK[17310] := 16#6D02;
   // UNICODE_TO_GBK[17311] := 16#9B90;
   // UNICODE_TO_GBK[17312] := 16#6D03;
   // UNICODE_TO_GBK[17313] := 16#9B91;
   // UNICODE_TO_GBK[17314] := 16#6D04;
   // UNICODE_TO_GBK[17315] := 16#E4A7;
   // UNICODE_TO_GBK[17316] := 16#6D05;
   // UNICODE_TO_GBK[17317] := 16#9B92;
   // UNICODE_TO_GBK[17318] := 16#6D06;
   // UNICODE_TO_GBK[17319] := 16#9B93;
   // UNICODE_TO_GBK[17320] := 16#6D07;
   // UNICODE_TO_GBK[17321] := 16#E4A6;
   // UNICODE_TO_GBK[17322] := 16#6D08;
   // UNICODE_TO_GBK[17323] := 16#9B94;
   // UNICODE_TO_GBK[17324] := 16#6D09;
   // UNICODE_TO_GBK[17325] := 16#9B95;
